(* Logix 5000 project; controller Safety vendor 1 type 14 code 86 rev 19.11; software revision 19.01 *)

TASK Periodic_0050ms (periodic, rate 50 ms, priority 11, watchdog 500 ms) : Comms
TASK SafetyTask (periodic, rate 50 ms, priority 10, watchdog 50 ms) : System, Estops, SafeOff

MODULES
   Local : vendor 1 type 14 code 86 (ICP 0, rev 19.11)
      Machine : vendor 1 type 14 code 96 (ICP 8, rev 19.13, $ae76c050$ RPI 20 ms)
      S16 : 1756-EN2T (Ethernet 192.168.1.200, ICP 16, rev 5.8)
      S2 : 1756-EN2T (ICP 2, Ethernet 192.168.1.10, rev 5.8, Input RPI 500 ms)
         SrDie_S1 : 1756-EN2T (Ethernet 192.168.1.18, rev 5.8)   // Shear Die Slot 01
            ShearDie : vendor 1 type 14 code 96 (ICP 0, rev 19.13, $8446c931$ RPI 20 ms)   // Shear Die Processor (Exit Section)
         CHPLC : 1734-AENTR (Ethernet 192.168.1.42, rev 3.10)
             : vendor 1 type 35 code 16 (PointIO 5, rev 1.1, Input RPI 50 ms, Output RPI 50 ms)
             : vendor 1 type 35 code 15 (PointIO 1, rev 1.1, Input RPI 50 ms)
             : vendor 1 type 35 code 15 (PointIO 3, rev 1.1, Input RPI 50 ms)
             : vendor 1 type 35 code 15 (PointIO 2, rev 1.1, Input RPI 50 ms)
             : vendor 1 type 35 code 16 (PointIO 6, rev 1.1, Input RPI 50 ms, Output RPI 50 ms)
             : vendor 1 type 35 code 16 (PointIO 4, rev 1.1, Output RPI 50 ms, Input RPI 50 ms)
         OS13 : 1734-AENTR (Ethernet 192.168.1.104, rev 3.10)
             : vendor 1 type 35 code 15 (PointIO 1, rev 1.1, Input RPI 50 ms)
         MCC2 : 1734-AENTR (Ethernet 192.168.1.41, rev 3.10)
             : vendor 1 type 35 code 16 (PointIO 1, rev 1.1, Output RPI 50 ms, Input RPI 10 ms)
             : vendor 1 type 35 code 16 (PointIO 2, rev 1.1, Input RPI 10 ms, Output RPI 50 ms)
         SDPLC : 1734-AENTR (Ethernet 192.168.1.79, rev 3.10)
             : vendor 1 type 35 code 15 (PointIO 1, rev 1.1, Input RPI 50 ms)
             : vendor 1 type 35 code 16 (PointIO 2, rev 1.1, Input RPI 50 ms, Output RPI 50 ms)
         MCC5 : 1734-AENTR (Ethernet 192.168.1.96, rev 3.10)
             : vendor 1 type 35 code 15 (PointIO 1, rev 1.1, Input RPI 10 ms)
             : vendor 1 type 35 code 16 (PointIO 5, rev 1.1, Input RPI 10 ms, Output RPI 50 ms)
             : vendor 1 type 35 code 16 (PointIO 3, rev 1.1, Input RPI 10 ms, Output RPI 50 ms)
             : vendor 1 type 35 code 16 (PointIO 4, rev 1.1, Input RPI 10 ms, Output RPI 50 ms)
         H1 : 1734-AENTR (Ethernet 192.168.1.120, rev 3.10)
             : vendor 1 type 35 code 15 (PointIO 6, rev 1.1, Input RPI 50 ms)
             : vendor 1 type 35 code 16 (PointIO 5, rev 1.1, Input RPI 50 ms, Output RPI 50 ms)
         G1 : 1734-AENTR (Ethernet 192.168.1.114, rev 3.10)
             : vendor 1 type 35 code 15 (PointIO 12, rev 1.1, Input RPI 50 ms)
             : vendor 1 type 35 code 16 (PointIO 11, rev 1.1, Input RPI 50 ms, Output RPI 50 ms)
         OS9 : 1734-AENTR (Ethernet 192.168.1.108, rev 3.10)
             : vendor 1 type 35 code 15 (PointIO 1, rev 1.1, Input RPI 50 ms)
         OS11 : 1734-AENTR (Ethernet 192.168.1.106, rev 3.10)
             : vendor 1 type 35 code 15 (PointIO 1, rev 1.1, Input RPI 50 ms)
         VS2 : 1734-AENTR (Ethernet 192.168.1.110, rev 3.10)
             : vendor 1 type 35 code 16 (PointIO 10, rev 1.1, Input RPI 50 ms, Output RPI 50 ms)
         OS16 : 1734-AENTR (Ethernet 192.168.1.97, rev 3.10)
             : vendor 1 type 35 code 15 (PointIO 1, rev 1.1, Input RPI 50 ms)
         OS8 : 1734-AENTR (Ethernet 192.168.1.116, rev 3.10)
             : vendor 1 type 35 code 15 (PointIO 1, rev 1.1, Input RPI 50 ms)
         E1 : 1734-AENTR (Ethernet 192.168.1.118, rev 3.10)
             : vendor 1 type 35 code 16 (PointIO 10, rev 1.1, Output RPI 50 ms, Input RPI 50 ms)
         DPD : 1734-AENTR (Ethernet 192.168.1.77, rev 3.10)
             : vendor 1 type 35 code 15 (PointIO 15, rev 1.1, Input RPI 50 ms)
             : vendor 1 type 35 code 16 (PointIO 14, rev 1.1, Input RPI 50 ms, Output RPI 50 ms)
         F1 : 1734-AENTR (Ethernet 192.168.1.112, rev 3.10)
             : vendor 1 type 35 code 15 (PointIO 20, rev 1.1, Input RPI 10 ms)
             : vendor 1 type 35 code 16 (PointIO 19, rev 1.1, Output RPI 50 ms, Input RPI 10 ms)
         OS14 : 1734-AENTR (Ethernet 192.168.1.102, rev 3.10)
             : vendor 1 type 35 code 15 (PointIO 1, rev 1.1, Input RPI 50 ms)
         MCC4 : 1734-AENTR (Ethernet 192.168.1.83, rev 3.10)
             : vendor 1 type 35 code 16 (PointIO 3, rev 1.1, Output RPI 50 ms, Input RPI 10 ms)
             : vendor 1 type 35 code 15 (PointIO 1, rev 1.1, Input RPI 10 ms)
             : vendor 1 type 35 code 16 (PointIO 4, rev 1.1, Output RPI 50 ms, Input RPI 10 ms)
         OS15 : 1734-AENTR (Ethernet 192.168.1.100, rev 3.10)
             : vendor 1 type 35 code 15 (PointIO 1, rev 1.1, Input RPI 50 ms)
      S3 : 1756-EN2T (Ethernet 192.168.1.11, ICP 3, rev 5.8, Input RPI 500 ms)
         OS3 : 1734-AENTR (Ethernet 192.168.1.40, rev 3.10)
             : vendor 1 type 35 code 15 (PointIO 1, rev 1.1, Input RPI 50 ms)
         OS1 : 1734-AENTR (Ethernet 192.168.1.70, rev 3.10)
             : vendor 1 type 35 code 15 (PointIO 1, rev 1.1, Input RPI 50 ms)
         D1 : 1734-AENTR (Ethernet 192.168.1.69, rev 3.10)
             : vendor 1 type 35 code 16 (PointIO 12, rev 1.1, Output RPI 50 ms, Input RPI 50 ms)
         OS4S : 1734-AENTR (Ethernet 192.168.1.57, rev 3.10)
             : vendor 1 type 35 code 16 (PointIO 5, rev 1.1, Input RPI 50 ms, Output RPI 50 ms)
             : vendor 1 type 35 code 15 (PointIO 1, rev 1.1, Input RPI 50 ms)
         OS5 : 1734-AENTR (Ethernet 192.168.1.62, rev 3.10)
             : vendor 1 type 35 code 15 (PointIO 1, rev 1.1, Input RPI 50 ms)
         A1 : 1734-AENTR (Ethernet 192.168.1.68, rev 3.10)
             : vendor 1 type 35 code 16 (PointIO 20, rev 1.1, Input RPI 50 ms, Output RPI 50 ms)
             : vendor 1 type 35 code 15 (PointIO 21, rev 1.1, Input RPI 50 ms)
         MCC3 : 1734-AENTR (Ethernet 192.168.1.38, rev 3.10)
             : vendor 1 type 35 code 16 (PointIO 4, rev 1.1, Input RPI 10 ms, Output RPI 50 ms)
             : vendor 1 type 35 code 16 (PointIO 3, rev 1.1, Input RPI 10 ms, Output RPI 50 ms)
             : vendor 1 type 35 code 15 (PointIO 1, rev 1.1, Input RPI 10 ms)
         MCC1 : 1734-AENTR (Ethernet 192.168.1.39, rev 3.10)
             : vendor 1 type 35 code 15 (PointIO 1, rev 1.1, Input RPI 10 ms)
             : vendor 1 type 35 code 16 (PointIO 6, rev 1.1, Input RPI 10 ms, Output RPI 50 ms)
         OS4N : 1734-AENTR (Ethernet 192.168.1.51, rev 3.10)
             : vendor 1 type 35 code 16 (PointIO 5, rev 1.1, Input RPI 50 ms, Output RPI 50 ms)
             : vendor 1 type 35 code 15 (PointIO 1, rev 1.1, Input RPI 50 ms)
         OS6 : 1734-AENTR (Ethernet 192.168.1.63, rev 3.10)
             : vendor 1 type 35 code 15 (PointIO 1, rev 1.1, Input RPI 50 ms)
         C1 : 1734-AENTR (Ethernet 192.168.1.43, rev 3.10)
             : vendor 1 type 35 code 16 (PointIO 12, rev 1.1, Output RPI 50 ms, Input RPI 10 ms)
         OS2 : 1734-AENTR (Ethernet 192.168.1.47, rev 3.10)
             : vendor 1 type 35 code 15 (PointIO 1, rev 1.1, Input RPI 50 ms)
      @b5ff5b04@:Partner : vendor 1 type 14 code 69 (ICP 1, rev 19.11)
END_MODULES

TYPE UDT_CardSts :
STRUCT
   EntrySts : DINT;   // Entry Status
   StandBy : BOOL;   // Stand By
   Faulted : BOOL;   // Faulted
   Validating : BOOL;   // Validating
   Connecting : BOOL;   // Connecting
   Running : BOOL;   // Running Connection OK
   ShuttingDown : BOOL;   // Shutting Down
   Inhibited : BOOL;   // Inhibited
   Waiting : BOOL;   // Waiting
END_STRUCT
END_TYPE

TYPE UDT_ShearStatus :
STRUCT
   Heartbeat : BOOL;   // Safety Status Heartbeat
   CoastStop : BOOL;   // Safety Status Coast Stop (0=Coast Stop) ( 1=OK)
   No_EStops : BOOL;   // Safety Status (0 = EStop) (1=OK)
   No_Faults : BOOL;   // Safety Status (1=No Faults)
   No_Motion : BOOL;   // Safety Status (1=No Motion)
   GuardsOK : BOOL;   // Safety Status Guards OK ( 1= OK)
   All_Drives_Off : BOOL;   // Safety Status All Drives Off (1=Off)
   ResetInput : BOOL;   // Safety Status Reset Input (1=Reset)
   FaultReset : BOOL;   // Safety Status (1=Fault Reset)
   CircuitReset : BOOL;   // Safety Status (1=Circuit Reset)
   CircuitResetTimer : TIMER;   // Safety Status Circuit Reset Timer
   StopTimer : TIMER;   // Safety Status Stop Timer Delay to Coast Drives
   BOOL : BOOL[32];   // Spare BOOLS
   DINT : DINT[5];   // Spare DINT
END_STRUCT
END_TYPE

TYPE UDT_SysStatus :
STRUCT
   Heartbeat : BOOL;   // Safety Status Heartbeat
   CoastStop_CTC : BOOL;   // Coil To Coil Safety Status Coast Stop (0=Coast Stop) ( 1=OK)
   CoastStop_CTL : BOOL;   // Cut To Length Safety Status Coast Stop (0=Coast Stop) ( 1=OK)
   CoastStop_Total : BOOL;   // Total Mode Safety Status Coast Stop (0=Coast Stop) ( 1=OK)
   No_CTC_EStops : BOOL;   // CTC Safety Status (0 = EStop) (1=OK)
   No_CTL_EStops : BOOL;   // CTL Safety Status (0 = EStop) (1=OK)
   No_Total_Estops : BOOL;   // Total Safety Status (0 = EStop) (1=OK)
   No_CTC_Faults : BOOL;   // Coil To Coil Safety Status (1=No Faults)
   No_CTL_Faults : BOOL;   // Cut To Length Safety Status (1=No Faults)
   No_Total_Faults : BOOL;   // Total Mode Safety Status (1=No Faults)
   No_Motion : BOOL;   // Safety Status (1=No Motion)
   GuardsOK : BOOL;   // Safety Status Guards OK ( 1= OK)
   All_Drives_Off : BOOL;   // Safety Status All Drives Off (1=Off)
   ResetInput_CTC : BOOL;   // Safety Status CTC Reset Input (1=Reset)
   ResetInput_CTL : BOOL;   // Safety Status CTL Reset Input (1=Reset)
   ResetInput_Total : BOOL;   // Safety Status Total Reset Input (1=Reset)
   FaultReset_CTC : BOOL;   // Safety Status CTC (1=Fault Reset)
   FaultReset_CTL : BOOL;   // Safety Status CTL (1=Fault Reset)
   FaultReset_Total : BOOL;   // Safety Status Total (1=Fault Reset)
   CircuitReset_CTC : BOOL;   // Safety Status CTC (1=Circuit Reset)
   CircuitReset_CTL : BOOL;   // Safety Status CTL (1=Circuit Reset)
   CircuitReset_Total : BOOL;   // Safety Status Total (1=Circuit Reset)
   CircuitResetTimer_CTC : TIMER;   // Safety Status Circuit Reset Timer
   CircuitResetTimer_CTL : TIMER;   // Safety Status CTL Circuit Reset Timer
   CircuitResetTimer_Total : TIMER;   // Safety Status Total Circuit Reset Timer
   CTCStopTimer : TIMER;   // Coil To Coil Safety Status Stop Timer Delay to Coast Drives
   CTLStopTimer : TIMER;   // Cut To Length Safety Status Stop Timer Delay to Coast Drives
   TotalStopTimer : TIMER;   // Total Mode Safety Status Stop Timer Delay to Coast Drives
   BOOL : BOOL[32];   // Spare BOOLS
   DINT : DINT[5];   // Spare DINT
END_STRUCT
END_TYPE

VAR_GLOBAL   (* controller tags *)
   A1_CoilCarSolPwrEn : BOOL;   // A1 UNW COIL CAR Solenoid Safe-Off Enable ( 1= Enable )
   A1_IO : UDT_CardSts[32] := ([0].EntrySts := 16897, [0].Running := 1);   // A1 Point I/O
        [4]   // 1734-IE2C/C
   A1_IOSts_Flt : BOOL;   // A1 Point IO Module Fault ( 1= Faulted)
   A1_S20_ModFlt : ALIAS FOR Flt_Modules[0].0;   // A1 Point I/O Slot20 Module Fault (1 = Fault)
   A1_S21_ModFlt : ALIAS FOR Flt_Modules[0].1;   // A1 Point I/O Slot21 Module Fault (1 = Fault)
   A1_SolPwrEn : BOOL := 1;   // A1 Solenoid Safe-Off Enable ( 1= Enable )
   A1_UnwLC_OK : BOOL := 1;   // Unwind Light Curtain A/B ( 1= Not Blocked) ( 0= Blocked)
   A1_UnwLC_RstCmd : BOOL;   // Unwind Light Curtain Reset Command ( 1= Reset Cmd)
   C1_IO : UDT_CardSts[32] := ([0].EntrySts := 16897, [0].Running := 1);   // C1 Point I/O
   C1_IOSts_Flt : BOOL;   // C1 Point IO Module Fault ( 1= Faulted)
   C1_S12_ModFlt : ALIAS FOR Flt_Modules[0].2;   // C1 Point I/O Slot12 Module Fault (1 = Fault)
   C1_SolPwrEn : BOOL := 1;   // C1 Solenoid Safe-Off Enable ( 1= Enable )
   CC : ALIAS FOR Diag_Tmp.0;   // Chris Como's Test Bit Always On Bit
   CC_Toggle : DINT := 4;   // TEST
   ChgMe : BOOL;
   ChgMe_x203PBL620 : BOOL;   // Need this from Machine OS1 Panel
   CHPLC_IO : UDT_CardSts[32] := ([0].EntrySts := 16897, [0].Running := 1);   // CHPLC Point I/O
   CHPLC_IOSts_Flt : BOOL;   // CHPLC Point IO Module Fault ( 1= Faulted)
   CHPLC_S1_ModFlt : ALIAS FOR Flt_Modules[0].3;   // CHPLC Point I/O Slot01 Module Fault (1 = Fault)
   CHPLC_S2_ModFlt : ALIAS FOR Flt_Modules[0].4;   // CHPLC Point I/O Slot02 Module Fault (1 = Fault)
   CHPLC_S3_ModFlt : ALIAS FOR Flt_Modules[0].5;   // CHPLC Point I/O Slot03 Module Fault (1 = Fault)
   CHPLC_S4_ModFlt : ALIAS FOR Flt_Modules[0].6;   // CHPLC Point I/O Slot04 Module Fault (1 = Fault)
   CHPLC_S5_ModFlt : ALIAS FOR Flt_Modules[0].7;   // CHPLC Point I/O Slot05 Module Fault (1 = Fault)
   CHPLC_S6_ModFlt : ALIAS FOR Flt_Modules[0].8;   // CHPLC Point I/O Slot06 Module Fault (1 = Fault)
   Citect_HB_Flt : BOOL;   // Citect Heartbeat Fault ( 1= Fault)
   Citect_HB_TOF : TIMER := (PRE := 2000, EN := 1, DN := 1);   // Citect Heartbeat Timer Off
   Citect_HB_TON : TIMER := (PRE := 2000, ACC := 850, EN := 1, TT := 1);   // Citect Heartbeat Timer On
   CommCards_OK : DINT := 30;   // Comm Cards OK
        .1   // Op Stations (Entry Section) Comm Cards OK ( 1= OK)
        .0   // MCC Comm Cards OK ( 1= OK)
        .2   // Op Stations (Exit Section) Comm Cards OK ( 1= OK)
        .3   // General I/O Comm Cards OK ( 1= OK)
        .4   // General I/O Comm Cards OK ( 1= OK)
        .31   // ALL Comm Cards OK ( 1= OK)
   D1_IO : UDT_CardSts[32] := ([0].EntrySts := 16897, [0].Running := 1);   // D1 Point I/O
        [4]   // 1734-IE2C/C
   D1_IOSts_Flt : BOOL;   // D1 Point IO Module Fault ( 1= Faulted)
   D1_S12_ModFlt : ALIAS FOR Flt_Modules[0].9;   // D1 Point I/O Slot12 Module Fault (1 = Fault)
   D1_SolPwrEn : BOOL := 1;   // D1 Solenoid Safe-Off Enable ( 1= Enable )
   DAM : ALIAS FOR Diag_Tmp.4;   // Doug M Always Off Test Bit
   Daniel_Ponstein_AFI : BOOL;
   Darin_M_Safety_Test_Bit : BOOL := 1;
   Darin_M_Test_Bit : DINT;
   DavidTest : BOOL;
   Diag_Tmp : DINT := 4079;   // Temp Bit Test Bit
        .17   // Temporary Test Bit: Logic 17
        .18   // Temporary Test Bit: Logic 18
        .0   // Temporary Test Bit 0: Logic 1
        .1   // Temporary Test Bit 1: Logic 1
        .10   // Temporary Test Bit: Logic 10
        .11   // Temporary Test Bit: Logic 11
        .12   // Temporary Test Bit: Logic 12
        .13   // Temporary Test Bit: Logic 13
        .14   // Temporary Test Bit: Logic 14
        .15   // Temporary Test Bit: Logic 15
        .16   // Temporary Test Bit: Logic 16
        .19   // Temporary Test Bit: Logic 19
        .2   // Temporary Test Bit 2: Logic 1
        .20   // Temporary Test Bit: Logic 20
        .21   // Temporary Test Bit: Logic 21
        .22   // Temporary Test Bit: Logic 22
        .23   // Temporary Test Bit: Logic 23
        .24   // Temporary Test Bit: Logic 24
        .25   // Temporary Test Bit: Logic 25
        .26   // Temporary Test Bit: Logic 26
        .27   // Temporary Test Bit: Logic 27
        .28   // Temporary Test Bit: Logic 28
        .29   // Temporary Test Bit: Logic 29
        .3   // Temporary Test Bit 3: Logic 1
        .30   // Temporary Test Bit: Logic 30
        .31   // Temporary Test Bit: Logic 31
        .4   // Temporary Test Bit 4: Logic 1
        .5   // Temporary Test Bit 5: Logic 1
        .6   // Temporary Test Bit 6: Logic 1
        .7   // Temporary Test Bit 6: Logic 1
        .8   // Temporary Test Bit: Logic 8
        .9   // Temporary Test Bit: Logic 9
   DPD_EstopRstCmd : BOOL;   // DPD Estop Reset Cmd
   DPD_FltRstCmd : BOOL;   // DPD Fault Reset Cmd
   DPD_IO : UDT_CardSts[32] := ([0].EntrySts := 16897, [0].Running := 1);   // DPD Point I/O
        [4]   // 1734-IE2C/C
   DPD_IOSts_Flt : BOOL;   // DPD Point IO Module Fault ( 1= Faulted)
   DPD_No_EStops : BOOL := 1;   // DPD No Estops ( 1= OK)
   DPD_S14_ModFlt : ALIAS FOR Flt_Modules[0].10;   // DPD Point I/O Slot14 Module Fault (1 = Fault)
   DPD_S15_ModFlt : ALIAS FOR Flt_Modules[0].11;   // DPD Point I/O Slot15 Module Fault (1 = Fault)
   DPD_SolPwrEn : BOOL := 1;   // DPD Solenoid Safe-Off Enable ( 1= Enable )
   Drives_Off : DINT;   // Line Drives Off
        .1   // Line AC Drives Off ( 1= Drvs Off)
        .0   // Line All DC Drives Off ( 1= Drvs Off)
        .4   // Shear Die Accelerator Drives Off ( 1= Drvs Off)
        .2   // Line AC Drives Off ( 1= Drvs Off)
        .3   // Line AC Drives Off ( 1= Drvs Off)
   E1_IO : UDT_CardSts[32] := ([0].EntrySts := 16897, [0].Running := 1);   // E1 Point I/O
        [4]   // 1734-IE2C/C
   E1_IOSts_Flt : BOOL;   // E1 Point IO Module Fault ( 1= Faulted)
   E1_S10_ModFlt : ALIAS FOR Flt_Modules[0].12;   // E1 Point I/O Slot10 Module Fault (1 = Fault)
   E1_SolPwrEn : BOOL := 1;   // E1 Solenoid Safe-Off Enable ( 1= Enable )
   EnBridle_DrvsOff : BOOL;   // Entry Bridle Drives OFF ( 1= OFF)
   EnBridle_SafeOffEn : BOOL := 1;   // Entry Bridle Safe-Off Enable ( 1= Enable )
   EnBridle_SafeOffFltRst : BOOL;   // Entry Bridle Safe-Off Fault Reset ( 1= Reset Cmd )
   ES_IndJog_PB : BOOL;   // Exit Section Individual Jog Select ( 1= Req Individual)
   ES_Line_JogPB : BOOL;   // Exit Section Line Jog PB ( 1= Ind Jog )
   ES_Line_RunPB : BOOL;   // Exit Section Line Run PB ( 1= Run)
   ES_Line_StopPB : BOOL := 1;   // Exit Section Line Stop PB ( 1= OK) (0=Stop)
   ES_Line_ThreadPB : BOOL;   // Exit Section Line Thread PB ( 1= Thread)
   ES_TndJog_PB : BOOL;   // Exit Section Tandem Jog PB (1= Tandem Jog Sel)
   ESTOP_x201PB040 : DCI_STOP := (ChannelA := 1, ChannelB := 1, InputStatus := 1, ColdStartType := 1, DiscrepancyTime := 250, O1 := 1);   // OS1 Line EStop Pushbutton
   ESTOP_x201PB040_Flt : ALIAS FOR Flt_Estops.0;   // OS1 Line EStop Pushbutton Fault ( 1= Fault)
   ESTOP_x211PB040 : DCI_STOP := (ChannelA := 1, ChannelB := 1, InputStatus := 1, ColdStartType := 1, DiscrepancyTime := 250, O1 := 1);   // OS2 Line EStop Pushbutton
   ESTOP_x211PB040_Flt : ALIAS FOR Flt_Estops.1;   // OS2 Line EStop Pushbutton Fault ( 1= Fault)
   ESTOP_x221PB040 : DCI_STOP := (ChannelA := 1, ChannelB := 1, InputStatus := 1, ColdStartType := 1, DiscrepancyTime := 250, O1 := 1);   // OS3 Line EStop Pushbutton
   ESTOP_x221PB040_Flt : ALIAS FOR Flt_Estops.2;   // OS3 Line EStop Pushbutton Fault ( 1= Fault)
   ESTOP_x231PB040 : DCI_STOP := (ChannelA := 1, ChannelB := 1, InputStatus := 1, ColdStartType := 1, DiscrepancyTime := 250, O1 := 1);   // OS4N Line EStop Pushbutton
   ESTOP_x231PB040_Flt : ALIAS FOR Flt_Estops.3;   // OS4N Line EStop Pushbutton Fault ( 1= Fault)
   ESTOP_x241PB040 : DCI_STOP := (ChannelA := 1, ChannelB := 1, InputStatus := 1, ColdStartType := 1, DiscrepancyTime := 250, O1 := 1);   // OS4S Line EStop Pushbutton
   ESTOP_x241PB040_Flt : ALIAS FOR Flt_Estops.4;   // OS4S Line EStop Pushbutton Fault ( 1= Fault)
   ESTOP_x251PB040 : DCI_STOP := (ChannelA := 1, ChannelB := 1, InputStatus := 1, ColdStartType := 1, DiscrepancyTime := 250, O1 := 1);   // OS5 Line EStop Pushbutton
   ESTOP_x251PB040_Flt : ALIAS FOR Flt_Estops.5;   // OS5 Line EStop Pushbutton Fault ( 1= Fault)
   ESTOP_x261PB040 : DCI_STOP := (ChannelA := 1, ChannelB := 1, InputStatus := 1, ColdStartType := 1, DiscrepancyTime := 250, O1 := 1);   // OS6 Line EStop Pushbutton
   ESTOP_x261PB040_Flt : ALIAS FOR Flt_Estops.6;   // OS6 Line EStop Pushbutton Fault ( 1= Fault)
   ESTOP_x271PB040 : DCI_STOP := (ChannelA := 1, ChannelB := 1, InputStatus := 1, ColdStartType := 1, DiscrepancyTime := 250, O1 := 1);   // OS8 Line EStop Pushbutton
   ESTOP_x271PB040_Flt : ALIAS FOR Flt_Estops.7;   // OS8 Line EStop Pushbutton Fault ( 1= Fault)
   ESTOP_x281PB040 : DCI_STOP := (ChannelA := 1, ChannelB := 1, InputStatus := 1, ColdStartType := 1, DiscrepancyTime := 250, O1 := 1);   // OS9 Line EStop Pushbutton
   ESTOP_x281PB040_Flt : ALIAS FOR Flt_Estops.8;   // OS9 Line EStop Pushbutton Fault ( 1= Fault)
   ESTOP_x291PB040 : DCI_STOP := (ChannelA := 1, ChannelB := 1, InputStatus := 1, ColdStartType := 1, DiscrepancyTime := 250, O1 := 1);   // OS11 Line EStop Pushbutton
   ESTOP_x291PB040_Flt : ALIAS FOR Flt_Estops.9;   // OS11 Line EStop Pushbutton Fault ( 1= Fault)
   ESTOP_x301PB040 : DCI_STOP := (ChannelA := 1, ChannelB := 1, InputStatus := 1, ColdStartType := 1, DiscrepancyTime := 250, O1 := 1);   // OS13 Line EStop Pushbutton
   ESTOP_x301PB040_Flt : ALIAS FOR Flt_Estops.10;   // OS13 Line EStop Pushbutton Fault ( 1= Fault)
   ESTOP_x311PB040 : DCI_STOP := (ChannelA := 1, ChannelB := 1, InputStatus := 1, ColdStartType := 1, DiscrepancyTime := 250, O1 := 1);   // OS14 Line EStop Pushbutton
   ESTOP_x311PB040_Flt : ALIAS FOR Flt_Estops.11;   // OS14 Line EStop Pushbutton Fault ( 1= Fault)
   ESTOP_x311PB130 : DCI_STOP := (ChannelA := 1, ChannelB := 1, InputStatus := 1, ColdStartType := 1, DiscrepancyTime := 250, O1 := 1);   // OS14 Shear Estop Pushbutton
   ESTOP_x311PB130_Flt : ALIAS FOR Flt_Estops.17;   // OS14 Shear EStop Pushbutton Fault ( 1= Fault)
   ESTOP_x321PB040 : DCI_STOP := (ChannelA := 1, ChannelB := 1, InputStatus := 1, ColdStartType := 1, DiscrepancyTime := 250, O1 := 1);   // OS15 Line EStop Pushbutton
   ESTOP_x321PB040_Flt : ALIAS FOR Flt_Estops.12;   // OS15 Line EStop Pushbutton Fault ( 1= Fault)
   ESTOP_x331PB040 : DCI_STOP := (ChannelA := 1, ChannelB := 1, InputStatus := 1, ColdStartType := 1, DiscrepancyTime := 250, O1 := 1);   // OS16 Line EStop Pushbutton
   ESTOP_x331PB040_Flt : ALIAS FOR Flt_Estops.13;   // OS16 Line EStop Pushbutton Fault ( 1= Fault)
   ESTOP_x480PB470 : DCI_STOP := (ChannelA := 1, ChannelB := 1, InputStatus := 1, ColdStartType := 1, DiscrepancyTime := 250, O1 := 1);   // DPD Line EStop Pushbutton
   ESTOP_x480PB470_Flt : ALIAS FOR Flt_Estops.14;   // DPD Line EStop Pushbutton Fault ( 1= Fault)
   ESTOP_x480PB550 : DCI_STOP := (ChannelA := 1, ChannelB := 1, InputStatus := 1, ColdStartType := 1, DiscrepancyTime := 250, O1 := 1);   // DPD (In Pit) Line EStop Pushbutton
   ESTOP_x480PB550_Flt : ALIAS FOR Flt_Estops.15;   // DPD Line EStop Pushbutton Fault ( 1= Fault)
   ESTOP_x519LS470 : DCI_STOP := (ChannelA := 1, ChannelB := 1, InputStatus := 1, ColdStartType := 1, DiscrepancyTime := 250, O1 := 1);   // G1 Tripwire Line EStop
   ESTOP_x519LS470_Flt : ALIAS FOR Flt_Estops.18;   // G1 Line EStop Tripwire Limit Switch Fault ( 1= Fault)
   ESTOP_x533PB470 : DCI_STOP := (ChannelA := 1, ChannelB := 1, InputStatus := 1, ColdStartType := 1, DiscrepancyTime := 250, O1 := 1);   // H1 Line EStop Pushbutton
   ESTOP_x533PB470_Flt : ALIAS FOR Flt_Estops.16;   // H1 Line EStop Pushbutton Fault ( 1= Fault)
   ExBridle_DrvsOff : BOOL;   // Exit Bridle Drives OFF ( 1= OFF)
   ExBridle_SafeOffEn : BOOL := 1;   // Exit Bridle Safe-Off Enable ( 1= Enable )
   ExBridle_SafeOffFltRst : BOOL;   // Exit Bridle Safe-Off Fault Reset ( 1= Reset Cmd )
   ExConHydPump_AutoStart : BOOL;   // (From Mach) Exit Conveyor Hydraulic Pump Auto Start Command
   F1_CoilCarSolPwrEn : BOOL := 1;   // F1 UNW COIL CAR Solenoid Safe-Off Enable ( 1= Enable )
   F1_IO : UDT_CardSts[32] := ([0].EntrySts := 16897, [0].Running := 1);   // F1 Point I/O
        [4]   // 1734-IE2C/C
   F1_IOSts_Flt : BOOL;   // F1 Point IO Module Fault ( 1= Faulted)
   F1_S19_ModFlt : ALIAS FOR Flt_Modules[0].13;   // F1 Point I/O Slot19 Module Fault (1 = Fault)
   F1_S20_ModFlt : ALIAS FOR Flt_Modules[0].14;   // F1 Point I/O Slot20 Module Fault (1 = Fault)
   F1_SolPwrEn : BOOL := 1;   // F1 Solenoid Safe-Off Enable ( 1= Enable )
   Flattener_FVR_En : BOOL := 1;   // Flattener FVR Enable ( 1= Enable )
   Flattener_FVR_FltRst : BOOL;   // Flattener Fault Reset ( 1= Reset Cmd )
   Flattener_FVR_FwdCmd : BOOL;   // Flattener Forward Command ( 1= Run Fwd )
   Flattener_FVR_RevCmd : BOOL;   // Flattener Reverse Command ( 1= Run Rev)
   Flt_Estops : DINT;   // Estop Fault Word
   Flt_Modules : DINT[5];   // Point IO Module Fault Word
   Flt_SafeOff : DINT[3];   // Safe Off Fault Word
   Flt_Starter : DINT;   // Starter Fault Word
   FltsToCitect : DINT[64];   // Faults to Citect
        [2]   // (Faults to Citect) Estop PB Faults
        [3]   // (Faults to Citect) Safe-Off Relay Faults
        [4]   // (Faults to Citect) FVR/FVNR Starter Faults
        [7]   // (Faults to Citect) MCC I/O Safety Module Faults
        [1]   // (Faults to Citect) Remote I/O Comm Faults
        [5]   // (Faults to Citect) General I/O Safety Module Faults
        [6]   // (Faults to Citect) Operator Station I/O Safety Module Faults
        [0].0   // Comm Loss Machine PLC
        [0].1   // Comm Loss Shear Die PLC
        [0].3   // Comm Loss Safety Slot 2
        [0].4   // Comm Loss Safety Slot 3
        [0].5   // Comm Loss Safety Slot 16
   FromCitect : DINT[64] := ([0] := 1, [10] := 22000, [11] := 22000, [12] := 12000, [13] := 12000, [14] := 12000);   // (From Citect)
        [1].10   // (From Citect)
        [1].12   // (From Citect)
        [1].13   // (From Citect)
        [1].14   // (From Citect)
        [1].15   // (From Citect)
        [1].16   // (From Citect)
        [1].11   // (From Citect)
        [0].19   // (From Citect)
        [0].0   // (From Citect) Heartbeat Reflected Back
        [0].1   // (From Citect) Exit Conveyor Hyd Pump Start
        [0].10   // (From Citect) Neg Tolerance Load PB
        [0].11   // (From Citect) Warning Count Load PB
        [0].12   // (From Citect) Scrap Length Load PB
        [0].13   // (From Citect) Scrap Reset PB
        [0].14   // (From Citect) Skid Count Load PB
        [0].15   // (From Citect) Shear Crank Start PB
        [0].16   // (From Citect) Shear Crank Stop PB
        [0].17   // (From Citect) Product Conveyors Start Command PB ( 1= Start)
        [0].18   // (From Citect) Product Conveyors Stop Command PB ( 1= Stop)
        [0].2   // (From Citect) Exit Conveyor Hyd Pump Stop
        [0].20   // (From Citect) Shear Pinch Roll Short Loop Select ( 1= Short Loop )
        [0].21   // (From Citect) Shear Pinch Roll Long Loop Select ( 1= Short Loop )
        [0].22   // (From Citect) Stacker Counter Reset PB
        [0].23   // (From Citect) Stacker Counter Increment PB
        [0].24   // (From Citect) Stacker Counter Decrement PB
        [0].25   // (From Citect) Good Piece Counter Reset PB
        [0].26   // (From Citect) Good Piece Counter Increment PB
        [0].27   // (From Citect) Good Piece Counter Decrement PB
        [0].28   // (From Citect) Lot Good Piece Counter Reset PB
        [0].29   // (From Citect) Lot Good Piece Counter Increment PB
        [0].3   // (From Citect) Sheeter Hyd Pump Start
        [0].30   // (From Citect) Lot Good Piece Counter Decrement PB
        [0].31   // (From Citect) Scrap Piece Counter Reset PB
        [0].4   // (From Citect) Sheeter Hyd Pump Stop
        [0].5   // (From Citect) Cut Length Load PB
        [0].6   // (From Citect) Cut Length Increase PB
        [0].7   // (From Citect) Cut Length Decrease PB
        [0].8   // (From Citect) Sheet Count Load PB
        [0].9   // (From Citect) Pos Tolerance Load PB
        [1].0   // (From Citect) Scrap Piece Counter Increment PB
        [1].1   // (From Citect) Scrap Piece Counter Decrement PB
        [1].17   // (From Citect)
        [1].18   // (From Citect)
        [1].19   // (From Citect)
        [1].2   // (From Citect) Home Position Set Command ( 1= Set Home Pos)
        [1].20   // (From Citect)
        [1].21   // (From Citect)
        [1].22   // (From Citect)
        [1].23   // (From Citect)
        [1].24   // (From Citect)
        [1].25   // (From Citect)
        [1].26   // (From Citect)
        [1].27   // (From Citect)
        [1].28   // (From Citect)
        [1].29   // (From Citect)
        [1].3   // (From Citect) Shear Lube Pump Start Command
        [1].30   // (From Citect)
        [1].31   // (From Citect)
        [1].4   // (From Citect) Shear Lube Pump Stop Command
        [1].5   // (From Citect) Sheeter Lube Pump Start Command
        [1].6   // (From Citect) Sheeter Lube Pump Stop Command
        [1].7   // (From Citect) Shear Metering Back Up Roll Light Gage Select
        [1].8   // (From Citect) Shear Metering Back Up Roll Heavy Gage Select
        [1].9   // (From Citect)
        [2].0   // (From Citect)
        [2].1   // (From Citect)
        [2].10   // (From Citect)
        [2].11   // (From Citect)
        [2].12   // (From Citect)
        [2].13   // (From Citect)
        [2].14   // (From Citect)
        [2].15   // (From Citect)
        [2].16   // (From Citect)
        [2].17   // (From Citect)
        [2].18   // (From Citect)
        [2].19   // (From Citect)
        [2].2   // (From Citect)
        [2].20   // (From Citect)
        [2].21   // (From Citect)
        [2].22   // (From Citect)
        [2].23   // (From Citect)
        [2].24   // (From Citect)
        [2].25   // (From Citect)
        [2].26   // (From Citect)
        [2].27   // (From Citect)
        [2].28   // (From Citect)
        [2].29   // (From Citect)
        [2].3   // (From Citect)
        [2].30   // (From Citect)
        [2].31   // (From Citect)
        [2].4   // (From Citect)
        [2].5   // (From Citect)
        [2].6   // (From Citect)
        [2].7   // (From Citect)
        [2].8   // (From Citect)
        [2].9   // (From Citect)
        [3]   // (From Citect) Set Scrap Length Inch
        [4]   // (From Citect) Warning Count
        [5]   // (From Citect) Next Cut Length Inch
        [6]   // (From Citect) Neg Tolerance Setpoint
        [7]   // (From Citect) Cut Length Inch
        [8]   // (From Citect) Skid Count Setpoint Pieces/Skid
        [9]   // (From Citect) Sheet Count Setpoint Pieces Before Warning
   FromMach : DINT[35];   // (FromMach)
   FromMachine : DINT[35] := ([0] := 164, [1] := 3, [3] := 16, [5] := 64, [10] := 50000, [11] := 100000, [12] := 1000000, [13] := 5000000, [15] := 3278258, [16] := 32, [19] := 44810, [21] := 44810);   // (FromMach)
        [0].1   // (FromMach) UWCC_Rst_PB Unwind Coil Car Safety Reset PB
        [0].24   // (FromMach)
        [0].25   // (FromMach)
        [0].7   // (FromMach)
        [0].4   // (FromMach)
        [0].3   // (FromMach)
        [0].0   // (FromMach) HB Heart Beat 0.25 Secs
        [0].19   // (FromMach)
        [0].20   // (FromMach)
        [0].21   // (FromMach)
        [0].23   // (FromMach)
        [0].18   // (FromMach)
        [0].8   // (FromMach)
        [0].9   // (FromMach)
        [0].16   // (FromMach)
        [0].17   // (FromMach)
        [0].22   // (FromMach)
        [0].5   // (FromMach)
        [0].10   // (FromMach) Hydraulic Pumps Auto Start Active
        [0].11   // (FromMach) Exit Conveyor Hydraulic Pump Auto Start Command
        [0].12   // (FromMach) Sheeter Hydraulic Pump Auto Start Command
        [0].13   // (FromMach) Lube Pumps Auto Start Active
        [0].14   // (FromMach) Sheeter PR Lube Pump Auto Start Command
        [0].15   // (FromMach) Shear PR Lube Pump Auto Start Command
        [0].26   // (FromMach)
        [0].27   // (FromMach)
        [0].28   // (FromMach)
        [0].29   // (FromMach)
        [0].30   // (FromMach)
        [0].31   // (FromMach)
        [1].0   // (FromMach)
        [1].1   // (FromMach)
        [1].2   // (FromMach)
        [1].3   // (FromMach)
        [1].4   // (FromMach)
        [1].5   // (FromMach)
        [1].6   // (FromMach)
        [1].7   // (FromMach)
        [1].8   // (FromMach)
        [1].9   // (FromMach)
        [1].10   // (FromMach)
        [1].11   // (FromMach)
        [1].12   // (FromMach)
        [1].13   // (FromMach)
        [1].14   // (FromMach)
        [1].15   // (FromMach)
        [1].16   // (FromMach)
        [1].17   // (FromMach)
        [1].18   // (FromMach)
        [1].19   // (FromMach)
        [1].20   // (FromMach)
        [1].21   // (FromMach)
        [1].22   // (FromMach)
        [1].23   // (FromMach)
        [1].24   // (FromMach)
        [1].25   // (FromMach)
        [1].26   // (FromMach)
        [1].27   // (FromMach)
        [1].28   // (FromMach)
        [1].29   // (FromMach)
        [1].30   // (FromMach)
        [1].31   // (FromMach)
        [2]   // (FromMach)
        [3]   // (FromMach)
        [4]   // (FromMach)
        [5].0   // (FromMach) Unwind Holddown Roll Jog Forward Command
        [5].1   // (FromMach) Unwind Holddown Roll Jog Reverse Command
        [5].2   // (FromMach) Flattener Jog Forward Command
        [5].3   // (FromMach) Flattener Jog Reverse Command
        [5].4   // (FromMach) Trimmer Pinch Roll Jog Forward Command
        [5].5   // (FromMach) Trimmer Pinch Roll Jog Reverse Command
        [5].6   // (FromMach) Trimmer Scrap Conveyor Jog Command
        [5].7   // (FromMach) Rewind Pinch Roll Jog Forward Command
        [5].8   // (FromMach) Rewind Pinch Roll Jog Reverse Command
        [5].9   // (FromMach)
        [5].10   // (FromMach)
        [5].11   // (FromMach)
        [5].12   // (FromMach)
        [5].13   // (FromMach)
        [5].14   // (FromMach)
        [5].15   // (FromMach)
        [5].16   // (FromMach)
        [5].17   // (FromMach)
        [5].18   // (FromMach)
        [5].19   // (FromMach)
        [5].20   // (FromMach)
        [5].21   // (FromMach)
        [5].22   // (FromMach)
        [5].23   // (FromMach)
        [5].24   // (FromMach)
        [5].25   // (FromMach)
        [5].26   // (FromMach)
        [5].27   // (FromMach)
        [5].28   // (FromMach)
        [5].29   // (FromMach)
        [5].30   // (FromMach)
        [5].31   // (FromMach)
        [0].6   // (FromMach) Line Emergency Stop Reset PBL
        [0].2   // (FromMach) Line TOTAL Mode ( 1= Total Mode) (0 = Coil to Coil)
   FromSafety : DINT[35] := ([0] := 16142, [1] := 14, [2] := 536870911, [4] := 64, [5] := 1); {produced}   // (From Safety)
        [2].30   // (From Safety)
        [0].0   // (From Safety) Heartbeat Pulse
        [5].0   // (From Safety) Shear Die Crank Running Fdbk ( 1= Running)
        [2].29   // (From Safety)
        [5].3   // (From Safety) Stacker Chain Fwd Fdbk
        [5].4   // (From Safety) Stacker Chain Rev Fdbk
        [5].1   // (From Safety) Scrap Horizontal Conveyor Fwd Fdbk
        [5].2   // (From Safety) Scrap Horizontal Conveyor Rev Fdbk
        [5].5   // (From Safety) Stacker Side Guide Lift Fwd Fdbk/Up
        [5].6   // (From Safety) Stacker Side Guide Lift Rev Fdbk/Down
        [4].3   // (From Safety) Flattener Drive Motor Rev Fdbk
        [1].1   // (From Safety) Shear Safety Status Coast Stop ( 0 = Coast Stop) ( 1= OK)
        [0].1   // (From Safety) Line Safety Status Coast Stop ( 0 = Coast Stop) ( 1= OK)
        [1].3   // (From Safety) Shear Safety Status No Faults ( 0 = Faults) ( 1= OK)
        [0].6   // (From Safety) Line Safety Status Guards OK ( 1= OK)
        [0]   // (From Safety)
        [0].8   // (From Safety)
        [0].4   // (From Safety)
        [0].9   // (From Safety)
        [0].7   // (From Safety)
        [2]   // (From Safety)
        [1].4   // (From Safety)
        [1].7   // (From Safety)
        [0].5   // (From Safety) Line Safety Status All Drives Off ( 1= All Off)
        [4].1   // (From Safety) Unwind Holddown Roll Drive Motor Rev Fdbk
        [0].2   // (From Safety) Line Safety Status EStop ( 0 = EStop) ( 1= OK)
        [0].3   // (From Safety) Line Safety Status No Faults ( 0 = Faults) ( 1= OK)
        [1].2   // (From Safety) Shear Safety Status EStop ( 0 = EStop) ( 1= OK)
        [1].5   // (From Safety) Shear Safety Status All Drives Off ( 1= All Off)
        [1].6   // (From Safety)
        [2].31   // (From Safety)
        [4].0   // (From Safety) Unwind Holddown Roll Drive Motor Fwd Fdbk
        [4].2   // (From Safety) Flattener Drive Motor Fwd Fdbk
        [4].4   // (From Safety) Trimmer Pinch Roll Fwd Fdbk
        [4].5   // (From Safety) Trimmer Pinch Roll Rev Fdbk
        [4].6   // (From Safety) Trimmer Scrap Conveyor RunFdbk
        [4].7   // (From Safety) Rewind Pinch Roll Fwd Fdbk
        [4].8   // (From Safety) Rewind Pinch Roll Rev Fdbk
        [2].0   // (From Safety) Unwind Op Side Drive Enable Relay
        [2].1   // (From Safety) Unwind Drive Side Drive Enable Relay
        [2].6   // (From Safety) Rewind Drive Enable Relay
        [2].9   // (From Safety) Paper Winder Safety Enable
        [2].12   // (From Safety) Scrap Choppers Safety Enable
        [2].22   // (From Safety) Shear Conveyor Safety Enable
        [2].27   // (From Safety) Stacker Blower Safety Enable
        [2].2   // (From Safety) #1 Entry Bridle Roll 2 Drive Enable Relay
        [2].3   // (From Safety) #2 Entry Bridle Roll 3 Drive Enable Relay
        [2].4   // (From Safety) #1 Exit Bridle Roll 6 Drive Enable Relay
        [2].5   // (From Safety) #2 Exit Bridle Roll 7 Drive Enable Relay
        [2].7   // (From Safety) Shear Die Drive Enable Relay
        [2].8   // (From Safety) Unwind Pinch Roll Safety Enable
        [2].10   // (From Safety) Trimmer Knives Width Adjust Safety Enable
        [2].11   // (From Safety) Trimmer Knives Safety Enable
        [2].13   // (From Safety) Scrap Choppers Width Adjust Safety Enable
        [2].14   // (From Safety) Washtank Pinch Roll 1 Safety Enable
        [2].15   // (From Safety) Washtank Pinch Roll 2 Safety Enable
        [2].16   // (From Safety) Washtank Pinch Roll 3 Safety Enable
        [2].17   // (From Safety) Washtank Pinch Roll 4 Safety Enable
        [2].18   // (From Safety) Side Guide Width Adjust Safety Enable
        [2].19   // (From Safety) Sheeter Pinch Roll Safety Enable
        [2].20   // (From Safety) Shear Pinch Roll Safety Enable
        [2].21   // (From Safety) Shear Metering Backup Roll Safety Enable
        [2].23   // (From Safety) Product Conveyor 1 Safety Enable
        [2].24   // (From Safety) Product Conveyor 2 Safety Enable
        [2].25   // (From Safety) Product Conveyor 3 Safety Enable
        [2].26   // (From Safety) Scrap Incline Conveyor Safety Enable
        [2].28   // (From Safety) Stacker Back Stop Safety Enable
   FromShearDie : DINT[35] := ([0] := 159, [1] := 8, [2] := 1056767, [5] := 1, [10] := 144000);   // (From Shear Die)
        [0].0   // (From Shear Die) Heartbeat Pulse
        [0].5   // (From Shear Die) Shear Emergency Stop Reset PBL
        [0].7   // (From Shear Die) Exit Section Line Stop PB ( 1= OK) (0=Stop)
        [0].10   // (From Shear Die) Exit Section Line Jog PB ( 1= Ind Jog)
        [5].3   // (From Shear Die) Stacker Chain Fwd Cmd
        [5].4   // (From Shear Die) Stacker Chain Rev Cmd
        [0].6   // (From Shear Die) Line Emergency Stop Reset PBL
        [0].4   // (From Shear DIe) Sheeter Pinch Roll Lube Run Fdbk
        [0].15   // (From Shear Die) Sheeter Pinch Roll Jog Forward SS
        [0].9   // (From Shear Die) Exit Section Line Thread PB ( 1= Thread)
        [0].8   // (From Shear Die) Exit Section Line Run PB ( 1= Run)
        [0].11   // (From Shear Die) Exit Section Tandem Jog PB (1= Tandem Jog Sel)
        [0].16   // (From Shear Die) Sheeter Pinch Roll Jog Reverse SS
        [0].1   // (From Shear DIe) Exit Conveyor Hyd Pump Run Fdbk
        [0].13   // (From Shear Die) Sheeter Pinch Roll Jog Forward SS
        [0].2   // (From Shear DIe) Sheeter Hyd Pump Run Fdbk
        [0].12   // (From Shear Die) Exit Section Individual Jog PB (1= Indiv Jog Sel)
        [0].18   // (From Shear Die) Shear Pinch Roll Jog Reverse SS
        [0].17   // (From Shear Die) Shear Pinch Roll Jog Forward SS
        [0].3   // (From Shear DIe) Shear Pinch Roll Lube Run Fdbk
        [0].14   // (From Shear Die) Sheeter Pinch Roll Jog Reverse SS
        [0].19   // (From Shear Die) Shear Conveyor Jog Forward SS
        [0].20   // (From Shear Die) Shear Conveyor Jog Reverse SS
        [0].21   // (From Shear Die) Product Conveyor Jog Forward PB
        [0].22   // (From Shear Die) Product Conveyor Jog Reverse PB
        [0].23   // (From Shear Die) Scrap Conveyor Jog Forward SS
        [0].24   // (From Shear Die) Scrap Conveyor Jog Reverse SS
        [1].0   // (From Shear Die) Scrap Mode Selected ( 1= Requested)
        [5].0   // (From Shear Die) Shear Die Crank Run Command ( 1= Run)
        [5].1   // (From Shear Die) Scrap Horizontal Conveyor Fwd Cmd ( 1= Run Fwd)
        [5].2   // (From Shear Die) Scrap Horizontal Conveyor Rev Cmd ( 1= Run Rev)
        [5].5   // (From Shear Die) Stacker Side Guide Lift Fwd Cmd/Up
        [5].6   // (From Shear Die) Stacker Side Guide Lift Rev Cmd/Dwn
   FUTURE : ALIAS FOR Diag_Tmp.1;   // FUTURE
   FVNR_y761MTR081RC : CONFIGURABLE_ROUT := (Actuate := 1, FeedbackType := 1, Feedback1 := 1, Feedback2 := 1, InputStatus := 1, OutputStatus := 1, FeedbackReactionTime := 250, O1 := 1, O2 := 1);   // Trimmer Scrap Conveyor FVNR Run Command
   FVNR_y778MTR080RC : CONFIGURABLE_ROUT := (Actuate := 1, FeedbackType := 1, Feedback1 := 1, Feedback2 := 1, InputStatus := 1, OutputStatus := 1, FeedbackReactionTime := 500, O1 := 1, O2 := 1);   // Shear Die Crank Motor FVNR Run Command
   FVR_y702MTR191_Flt : ALIAS FOR Flt_Starter.4;   // Rewind Pinch Roll Starter Fault ( 1= Fault)
   FVR_y702MTR191FC : CONFIGURABLE_ROUT := (FeedbackType := 1, InputStatus := 1, OutputStatus := 1, FeedbackReactionTime := 1000);   // Rewind Pinch Roll FVR Fwd Command
   FVR_y702MTR191RC : CONFIGURABLE_ROUT := (FeedbackType := 1, InputStatus := 1, OutputStatus := 1, FeedbackReactionTime := 1000);   // Rewind Pinch Roll FVR Rev Command
   FVR_y708MTR080_Flt : ALIAS FOR Flt_Starter.1;   // Flattener Drive Motor Starter Fault ( 1= Fault)
   FVR_y708MTR080FC : CONFIGURABLE_ROUT := (FeedbackType := 1, InputStatus := 1, OutputStatus := 1, FeedbackReactionTime := 250);   // Flattener Drive Motor FVR Fwd Command
   FVR_y708MTR080RC : CONFIGURABLE_ROUT := (FeedbackType := 1, InputStatus := 1, OutputStatus := 1, FeedbackReactionTime := 250);   // Flattener Drive Motor FVR Rev Command
   FVR_y708MTR250_Flt : ALIAS FOR Flt_Starter.0;   // Unwind Hold Down Roll Starter Fault ( 1= Fault)
   FVR_y708MTR250FC : CONFIGURABLE_ROUT := (FeedbackType := 1, InputStatus := 1, OutputStatus := 1, FeedbackReactionTime := 250);   // Unwind Hold Down Roll FVR Fwd Command
   FVR_y708MTR250RC : CONFIGURABLE_ROUT := (FeedbackType := 1, InputStatus := 1, OutputStatus := 1, FeedbackReactionTime := 250);   // Unwind Hold Down Roll FVR Rev Command
   FVR_y753MTR190_Flt : ALIAS FOR Flt_Starter.2;   // Trimmer Pinch Roll Starter Fault ( 1= Fault)
   FVR_y753MTR190FC : CONFIGURABLE_ROUT := (FeedbackType := 1, InputStatus := 1, OutputStatus := 1, FeedbackReactionTime := 250);   // Trimmer Pinch Roll FVR Fwd Command
   FVR_y753MTR190RC : CONFIGURABLE_ROUT := (FeedbackType := 1, InputStatus := 1, OutputStatus := 1, FeedbackReactionTime := 250);   // Trimmer Pinch Roll FVR Rev Command
   FVR_y761MTR081_Flt : ALIAS FOR Flt_Starter.3;   // Trimmer Scrap Conveyor Starter Fault ( 1= Fault)
   FVR_y778MTR080_Flt : ALIAS FOR Flt_Starter.5;   // Shear Die Crank Starter Fault ( 1= Fault)
   FVR_y802MTR080_Flt : ALIAS FOR Flt_Starter.6;   // Stacker Side Guide Lift Starter Fault ( 1= Fault)
   FVR_y802MTR080FC : CONFIGURABLE_ROUT := (FeedbackType := 1, InputStatus := 1, OutputStatus := 1, FeedbackReactionTime := 250);   // Stacker Side Guide Lift FVR Fwd Command
   FVR_y802MTR080RC : CONFIGURABLE_ROUT := (FeedbackType := 1, InputStatus := 1, OutputStatus := 1, FeedbackReactionTime := 250);   // Stacker Side Guide Lift FVR Rev Command
   FVR_y802MTR230_Flt : ALIAS FOR Flt_Starter.8;   // Scrap Horizontal Conveyor Starter Fault ( 1= Fault)
   FVR_y802MTR230FC : CONFIGURABLE_ROUT := (FeedbackType := 1, InputStatus := 1, OutputStatus := 1, FeedbackReactionTime := 250);   // Scrap Horizontal Conveyor FVR Fwd Command
   FVR_y802MTR230RC : CONFIGURABLE_ROUT := (FeedbackType := 1, InputStatus := 1, OutputStatus := 1, FeedbackReactionTime := 250);   // Scrap Horizontal Conveyor FVR Rev Command
   FVR_y802MTR231_Flt : ALIAS FOR Flt_Starter.7;   // Stacker Chain Conveyor Starter Fault ( 1= Fault)
   FVR_y802MTR231FC : CONFIGURABLE_ROUT := (FeedbackType := 1, InputStatus := 1, OutputStatus := 1, FeedbackReactionTime := 250);   // Stacker Chain Conveyor FVR Fwd Command
   FVR_y802MTR231RC : CONFIGURABLE_ROUT := (FeedbackType := 1, InputStatus := 1, OutputStatus := 1, FeedbackReactionTime := 250);   // Stacker Chain Conveyor FVR Rev Command
   G1_EstopRstCmd : BOOL;   // G1 Estop Reset Command ( 1= Reset Cmd)
   G1_FltRstCmd : BOOL;   // G1 Fault Reset Command ( 1= Reset Cmd)
   G1_IO : UDT_CardSts[32] := ([0].EntrySts := 16897, [0].Running := 1);   // G1 Point I/O
        [4]   // 1734-IE2C/C
   G1_IOSts_Flt : BOOL;   // G1 Point IO Module Fault ( 1= Faulted)
   G1_No_EStops : BOOL := 1;   // G1 No Estops ( 1= OK)
   G1_S11_ModFlt : ALIAS FOR Flt_Modules[0].15;   // G1 Point I/O Slot11 Module Fault (1 = Fault)
   G1_S12_ModFlt : ALIAS FOR Flt_Modules[0].16;   // G1 Point I/O Slot12 Module Fault (1 = Fault)
   G1_SolPwrEn : BOOL := 1;   // G1 Solenoid Safe-Off Enable ( 1= Enable )
   H1_EstopRstCmd : BOOL;   // H1 Estop Reset Command ( 1= Reset Cmd)
   H1_FltRstCmd : BOOL;   // H1 Fault Reset Command ( 1= Reset Cmd)
   H1_IO : UDT_CardSts[32] := ([0].EntrySts := 16897, [0].Running := 1);   // H1 Point I/O
        [4]   // 1734-IE2C/C
   H1_IOSts_Flt : BOOL;   // H1 Point IO Module Fault ( 1= Faulted)
   H1_No_EStops : BOOL := 1;   // H1 No Estops ( 1= OK)
   H1_S5_ModFlt : ALIAS FOR Flt_Modules[0].17;   // H1 Point I/O Slot05 Module Fault (1 = Fault)
   H1_S6_ModFlt : ALIAS FOR Flt_Modules[0].18;   // H1 Point I/O Slot06 Module Fault (1 = Fault)
   H1_SolPwrEn : BOOL := 1;   // H1 Solenoid Safe-Off Enable ( 1= Enable )
   HB_Citect : BOOL := 1;   // Heartbeat Citect Reflect
   HydPumps_AutoStart : BOOL;   // (From Mach) Hydraulic Pumps Auto Start Active
   IOCards_OK : DINT;   // Point I/O Cards OK
        .0   // MCC I/O Cards OK ( 1= OK)
        .1   // Op Stations (Entry Section) I/O Cards OK ( 1= OK)
        .2   // Op Stations (Exit Section) I/O Cards OK ( 1= OK)
        .3   // General I/O I/O Cards OK ( 1= OK)
        .4   // General I/O I/O Cards OK ( 1= OK)
        .31   // ALL I/O Cards OK ( 1= OK)
   jay : BOOL := 1;
   Line_CTC_CoastStop : BOOL;   // Line Coast Stop ( 1= Coast Stop) (Condition Exists)
   Line_CTL_CoastStop : BOOL;   // Line Coast Stop ( 1= Coast Stop) (Condition Exists)
   Line_No_Estop : DINT := -2147483645;   // Line Estop Summation ( 1= No Estop PB's) (Pressed)
   Line_NoP2P_CommFlts : BOOL := 1;   // Line No Peer to Peer Comm Faults ( 1= OK)
   Line_Total_CoastStop : BOOL;   // Line Coast Stop ( 1= Coast Stop) (Condition Exists)
   Line_TotalMode : BOOL := 1;   // Line TOTAL Mode ( 1= Total Mode) (0 = Coil to Coil)
   LineSts : UDT_SysStatus := (Heartbeat := 1, CoastStop_CTC := 1, CoastStop_CTL := 1, CoastStop_Total := 1, No_CTC_EStops := 1, No_CTL_EStops := 1, No_Total_Estops := 1, No_CTC_Faults := 1, No_CTL_Faults := 1, No_Total_Faults := 1, CTCStopTimer.PRE := 5000, CTLStopTimer.PRE := 5000, TotalStopTimer.PRE := 5000);
   Local_ModFlts : DINT := 514;   // Local Card Fault Status
        .1   // Slot 01
        .2   // Slot 02 1756-EN2T Card Fault ( 1= Fault)
        .3   // Slot 03 1756-EN2T Card Fault ( 1= Fault)
        .9   // Slot 09
        .16   // Slot 16 1756-EN2T Card Fault ( 1= Fault)
   Local_Networks_OK : BOOL := 1;   // Local Network CARDS OK ( 1= OK)
   Local_Slot : UDT_CardSts[17] := ([1].EntrySts := 24576, [2].EntrySts := 16897, [2].Running := 1, [3].EntrySts := 16897, [3].Running := 1, [4].EntrySts := 16897, [4].Running := 1, [5].EntrySts := 16897, [5].Running := 1, [6].EntrySts := 16897, [6].Running := 1, [7].EntrySts := 16897, [7].Running := 1, [9].EntrySts := 24576, [16].EntrySts := 16897, [16].Running := 1); {access Read Only}   // Safety Processor
        [8]   // 1756-L75 -
        [2]   // 1756-EN2T -
        [3]   // 1756-EN2T -
        [16]   // 1756-EN2T -
   LubePumps_AutoStart : BOOL;   // (From Mach) Lube Pumps Auto Start Active
   Machine_HB_Flt : BOOL;   // Machine Heartbeat Fault ( 1= Fault)
   Machine_HB_TOF : TIMER := (PRE := 1000);   // Machine Heartbeat Timer Off
   Machine_HB_TON : TIMER := (PRE := 1000, ACC := 100, EN := 1, TT := 1);   // Machine Heartbeat Timer On
   Map_Citect : DINT[5] := ([0] := 1);   // Mapped From Shear Citect System
        [0].0   // Citect Heartbeat Fault ( 1= Fault)
   Map_Mach : DINT[5] := ([0] := 4225);   // From Machine Processor
        [0].0   // (From Machine) Heartbeat Pulse
        [0].1   // Unwind Hold Down Roll Forward Command ( 1= Run Fwd )
        [0].2   // Unwind Hold Down Roll Reverse Command ( 1= Run Rev)
        [0].3   // Flattener Forward Command ( 1= Run Fwd )
        [0].4   // Flattener Reverse Command ( 1= Run Rev)
        [0].5   // Trimmer Pinch Roll Forward Command ( 1= Run Fwd )
        [0].6   // Trimmer Pinch Roll Reverse Command ( 1= Run Rev)
        [0].7   // Trimmer Scrap Conveyor Run Command ( 1= Run )
        [0].8   // Rewind Pinch Roll Forward Command ( 1= Run Fwd )
        [0].9   // Rewind Pinch Roll Reverse Command ( 1= Run Rev)
        [0].10   // Unwind Coil Car Safety Reset PB
        [0].11   // Line Emergency Stop Reset PBL
        [0].12   // Line TOTAL Mode ( 1= Total Mode) (0 = Coil to Coil)
   Map_ShDie : DINT[5] := ([0] := 3);   // Mapped From Shear Die Processor
        [0].1   // Shear Die Crank Run Command ( 1= Run)
        [0].2   // Scrap Horizontal Conveyor Fwd Cmd ( 1= Run Fwd)
        [0].3   // Scrap Horizontal Conveyor Rev Cmd ( 1= Run Rev)
        [0].4   // Stacker Chain Fwd Cmd
        [0].5   // Stacker Chain Rev Cmd
        [0].7   // Stacker Side Guide Lift Rev Cmd/Dwn
        [0].6   // Stacker Side Guide Lift Fwd Cmd/Up
        [0].8   // Shear Emergency Stop Reset PBL
        [0].0   // (From Shear Die) Heartbeat Pulse
        [0].9   // Line Emergency Stop Reset PBL
   MCC1_IO : UDT_CardSts[32] := ([0].EntrySts := 16897, [0].Running := 1);   // MCC1 Point I/O
        [13]   // 1734-IE2V/C
   MCC1_IOSts_Flt : BOOL;   // MCC1 Point IO Module Fault ( 1= Faulted)
   MCC1_S1_ModFlt : ALIAS FOR Flt_Modules[2].0;   // MCC1 Point I/O Slot01 Module Fault (1 = Fault)
   MCC1_S6_ModFlt : ALIAS FOR Flt_Modules[2].1;   // MCC1 Point I/O Slot06 Module Fault (1 = Fault)
   MCC2_IO : UDT_CardSts[32] := ([0].EntrySts := 28928);   // MCC2 Point I/O
        [13]   // 1734-IE2V/C
   MCC2_IOSts_Flt : BOOL;   // MCC2 Point IO Module Fault ( 1= Faulted)
   MCC2_S1_ModFlt : ALIAS FOR Flt_Modules[2].2;   // MCC2 Point I/O Slot01 Module Fault (1 = Fault)
   MCC2_S2_ModFlt : ALIAS FOR Flt_Modules[2].3;   // MCC2 Point I/O Slot02 Module Fault (1 = Fault)
   MCC3_IO : UDT_CardSts[32] := ([0].EntrySts := 16897, [0].Running := 1);   // MCC3 Point I/O
   MCC3_IOSts_Flt : BOOL;   // MCC3 Point IO Module Fault ( 1= Faulted)
   MCC3_S1_ModFlt : ALIAS FOR Flt_Modules[2].4;   // MCC3 Point I/O Slot01 Module Fault (1 = Fault)
   MCC3_S3_ModFlt : ALIAS FOR Flt_Modules[2].5;   // MCC3 Point I/O Slot03 Module Fault (1 = Fault)
   MCC3_S4_ModFlt : ALIAS FOR Flt_Modules[2].6;   // MCC3 Point I/O Slot04 Module Fault (1 = Fault)
   MCC4_IO : UDT_CardSts[32] := ([0].EntrySts := 16897, [0].Running := 1);   // MCC4 Point I/O
   MCC4_IOSts_Flt : BOOL;   // MCC-4 Point IO Module Fault ( 1= Faulted)
   MCC4_S1_ModFlt : ALIAS FOR Flt_Modules[2].7;   // MCC4 Point I/O Slot01 Module Fault (1 = Fault)
   MCC4_S3_ModFlt : ALIAS FOR Flt_Modules[2].8;   // MCC4 Point I/O Slot03 Module Fault (1 = Fault)
   MCC4_S4_ModFlt : ALIAS FOR Flt_Modules[2].9;   // MCC4 Point I/O Slot04 Module Fault (1 = Fault)
   MCC5_IO : UDT_CardSts[32] := ([0].EntrySts := 28928);   // MCC5 Point I/O
   MCC5_IOSts_Flt : BOOL;   // MCC-5 Point IO Module Fault ( 1= Faulted)
   MCC5_S1_ModFlt : ALIAS FOR Flt_Modules[2].10;   // MCC5 Point I/O Slot01 Module Fault (1 = Fault)
   MCC5_S3_ModFlt : ALIAS FOR Flt_Modules[2].11;   // MCC5 Point I/O Slot03 Module Fault (1 = Fault)
   MCC5_S4_ModFlt : ALIAS FOR Flt_Modules[2].12;   // MCC5 Point I/O Slot04 Module Fault (1 = Fault)
   MCC5_S5_ModFlt : ALIAS FOR Flt_Modules[2].13;   // MCC5 Point I/O Slot05 Module Fault (1 = Fault)
   OS11_EstopRstCmd : BOOL;   // OS11 Estop Reset Command ( 1= Reset Cmd)
   OS11_FltRstCmd : BOOL;   // OS11 Fault Reset Command ( 1= Reset Cmd)
   OS11_IO : UDT_CardSts[32] := ([0].EntrySts := 16897, [0].Running := 1);   // OS11 Point I/O
        [4]   // 1734-IE2C/C
   OS11_IOSts_Flt : BOOL;   // OS11 Point IO Module Fault ( 1= Faulted)
   OS11_No_EStops : BOOL := 1;   // OS11 No Estops ( 1= OK)
   OS11_S1_ModFlt : ALIAS FOR Flt_Modules[1].11;   // OS11 Point I/O Slot01 Module Fault (1 = Fault)
   OS13_EstopRstCmd : BOOL;   // OS13 Estop Reset Command ( 1= Reset Cmd)
   OS13_FltRstCmd : BOOL;   // OS13 Fault Reset Command ( 1= Reset Cmd)
   OS13_IO : UDT_CardSts[32] := ([0].EntrySts := 16897, [0].Running := 1);   // OS13 Point I/O
        [4]   // 1734-IE2C/C
   OS13_IOSts_Flt : BOOL;   // OS13 Point IO Module Fault ( 1= Faulted)
   OS13_No_EStops : BOOL := 1;   // OS13 No Estops ( 1= OK)
   OS13_S1_ModFlt : ALIAS FOR Flt_Modules[1].12;   // OS13 Point I/O Slot01 Module Fault (1 = Fault)
   OS14_EstopRstCmd : BOOL;   // OS14 Estop Reset Command ( 1= Reset Cmd)
   OS14_FltRstCmd : BOOL;   // OS14 Fault Reset Command ( 1= Reset Cmd)
   OS14_IO : UDT_CardSts[32] := ([0].EntrySts := 16897, [0].Running := 1);   // OS14 Point I/O
        [13]   // 1734-IE2V/C
   OS14_IOSts_Flt : BOOL;   // OS14 Point IO Module Fault ( 1= Faulted)
   OS14_No_EStops : BOOL := 1;   // OS14 No Estops ( 1= OK)
   OS14_S1_ModFlt : ALIAS FOR Flt_Modules[1].13;   // OS14 Point I/O Slot01 Module Fault (1 = Fault)
   OS14_Shear_EstopRstCmd : BOOL;   // OS14_Shear Estop Reset Command ( 1= Reset Cmd)
   OS14_Shear_FltRstCmd : BOOL;   // OS14_Shear Fault Reset Command ( 1= Reset Cmd)
   OS14_Shear_No_EStops : BOOL := 1;   // OS14_Shear No Estops ( 1= OK)
   OS15_EstopRstCmd : BOOL;   // OS15 Estop Reset Command ( 1= Reset Cmd)
   OS15_FltRstCmd : BOOL;   // OS15 Fault Reset Command ( 1= Reset Cmd)
   OS15_IO : UDT_CardSts[32] := ([0].EntrySts := 16897, [0].Running := 1);   // OS15 Point I/O
   OS15_IOSts_Flt : BOOL;   // OS15 Point IO Module Fault ( 1= Faulted)
   OS15_No_EStops : BOOL := 1;   // OS15 No Estops ( 1= OK)
   OS15_S1_ModFlt : ALIAS FOR Flt_Modules[1].14;   // OS15 Point I/O Slot01 Module Fault (1 = Fault)
   OS16_EstopRstCmd : BOOL;   // OS16 Estop Reset Command ( 1= Reset Cmd)
   OS16_FltRstCmd : BOOL;   // OS16 Fault Reset Command ( 1= Reset Cmd)
   OS16_IO : UDT_CardSts[32] := ([0].EntrySts := 16897, [0].Running := 1);   // OS16 Point I/O
   OS16_IOSts_Flt : BOOL;   // OS16 Point IO Module Fault ( 1= Faulted)
   OS16_No_EStops : BOOL := 1;   // OS16 No Estops ( 1= OK)
   OS16_S1_ModFlt : ALIAS FOR Flt_Modules[1].15;   // OS16 Point I/O Slot01 Module Fault (1 = Fault)
   OS1_EstopRstCmd : BOOL;   // OS1 Estop Reset Command ( 1= Reset Cmd)
   OS1_FltRstCmd : BOOL;   // OS1 Fault Reset Command ( 1= Reset Cmd)
   OS1_IO : UDT_CardSts[32] := ([0].EntrySts := 16897, [0].Running := 1);   // OS1 Point I/O
        [4]   // 1734-IE2C/C
   OS1_IOSts_Flt : BOOL;   // OS1 Point IO Module Fault ( 1= Faulted)
   OS1_No_EStops : BOOL := 1;   // OS1 No Estops ( 1= OK)
   OS1_S1_ModFlt : ALIAS FOR Flt_Modules[1].0;   // OS1 Point I/O Slot01 Module Fault (1 = Fault)
   OS2_EstopRstCmd : BOOL;   // OS2 Estop Reset Command ( 1= Reset Cmd)
   OS2_FltRstCmd : BOOL;   // OS2 Fault Reset Command ( 1= Reset Cmd)
   OS2_IO : UDT_CardSts[32] := ([0].EntrySts := 16897, [0].Running := 1, [1].EntrySts := 16897, [1].Running := 1, [3].EntrySts := 16899, [3].Running := 1, [4].EntrySts := 16897, [4].Running := 1, [5].EntrySts := 16897, [5].Running := 1, [6].EntrySts := 16897, [6].Running := 1, [7].EntrySts := 16897, [7].Running := 1); {access Read Only}   // OS2 Point I/O
   OS2_IOSts_Flt : BOOL;   // OS2 Point IO Module Fault ( 1= Faulted)
   OS2_No_EStops : BOOL := 1;   // OS2 No Estops ( 1= OK)
   OS2_S1_ModFlt : ALIAS FOR Flt_Modules[1].1;   // OS2 Point I/O Slot01 Module Fault (1 = Fault)
   OS3_EstopRstCmd : BOOL;   // OS3 Estop Reset Command ( 1= Reset Cmd)
   OS3_FltRstCmd : BOOL;   // OS3 Fault Reset Command ( 1= Reset Cmd)
   OS3_IO : UDT_CardSts[32] := ([0].EntrySts := 16897, [0].Running := 1);   // OS3 Point I/O
   OS3_IOSts_Flt : BOOL;   // OS3 Point IO Module Fault ( 1= Faulted)
   OS3_No_EStops : BOOL := 1;   // OS3 No Estops ( 1= OK)
   OS3_S1_ModFlt : ALIAS FOR Flt_Modules[1].2;   // OS3 Point I/O Slot01 Module Fault (1 = Fault)
   OS4_EstopRstCmd : BOOL;   // OS4 Estop Reset Command ( 1= Reset Cmd)
   OS4_FltRstCmd : BOOL;   // OS4 Fault Reset Command ( 1= Reset Cmd)
   OS4_No_EStops : BOOL := 1;   // OS4 No Estops ( 1= OK)
   OS4N_IO : UDT_CardSts[32] := ([0].EntrySts := 16897, [0].Running := 1);   // OS4N Point I/O
        [4]   // 1734-IE2C/C
   OS4N_IOSts_Flt : BOOL;   // OS4N Point IO Module Fault ( 1= Faulted)
   OS4N_S1_ModFlt : ALIAS FOR Flt_Modules[1].3;   // OS4N Point I/O Slot01 Module Fault (1 = Fault)
   OS4N_S5_ModFlt : ALIAS FOR Flt_Modules[1].4;   // OS4N Point I/O Slot05 Module Fault (1 = Fault)
   OS4N_SolPwrEn : BOOL := 1;   // OS4N Solenoid Safe-Off Enable ( 1= Enable )
   OS4S_IO : UDT_CardSts[32] := ([0].EntrySts := 16897, [0].Running := 1);   // OS4S Point I/O
        [4]   // 1734-IE2C/C
   OS4S_IOSts_Flt : BOOL;   // OS4S Point IO Module Fault ( 1= Faulted)
   OS4S_S1_ModFlt : ALIAS FOR Flt_Modules[1].5;   // OS4S Point I/O Slot01 Module Fault (1 = Fault)
   OS4S_S5_ModFlt : ALIAS FOR Flt_Modules[1].6;   // OS4S Point I/O Slot05 Module Fault (1 = Fault)
   OS4S_SolPwrEn : BOOL := 1;   // OS4S Solenoid Safe-Off Enable ( 1= Enable )
   OS5_EstopRstCmd : BOOL;   // OS5 Estop Reset Command ( 1= Reset Cmd)
   OS5_FltRstCmd : BOOL;   // OS5 Fault Reset Command ( 1= Reset Cmd)
   OS5_IO : UDT_CardSts[32] := ([0].EntrySts := 16897, [0].Running := 1);   // OS5 Point I/O
        [4]   // 1734-IE2C/C
   OS5_IOSts_Flt : BOOL;   // OS5 Point IO Module Fault ( 1= Faulted)
   OS5_No_EStops : BOOL := 1;   // OS5 No Estops ( 1= OK)
   OS5_S1_ModFlt : ALIAS FOR Flt_Modules[1].7;   // OS5 Point I/O Slot01 Module Fault (1 = Fault)
   OS6_EstopRstCmd : BOOL;   // OS6 Estop Reset Command ( 1= Reset Cmd)
   OS6_FltRstCmd : BOOL;   // OS6 Fault Reset Command ( 1= Reset Cmd)
   OS6_IO : UDT_CardSts[32] := ([0].EntrySts := 16897, [0].Running := 1);   // OS6 Point I/O
        [4]   // 1734-IE2C/C
   OS6_IOSts_Flt : BOOL;   // OS6 Point IO Module Fault ( 1= Faulted)
   OS6_No_EStops : BOOL := 1;   // OS6 No Estops ( 1= OK)
   OS6_S1_ModFlt : ALIAS FOR Flt_Modules[1].8;   // OS6 Point I/O Slot01 Module Fault (1 = Fault)
   OS8_EstopRstCmd : BOOL;   // OS8 Estop Reset Command ( 1= Reset Cmd)
   OS8_FltRstCmd : BOOL;   // OS8 Fault Reset Command ( 1= Reset Cmd)
   OS8_IO : UDT_CardSts[32] := ([0].EntrySts := 16897, [0].Running := 1);   // OS8 Point I/O
        [4]   // 1734-IE2C/C
   OS8_IOSts_Flt : BOOL;   // OS8 Point IO Module Fault ( 1= Faulted)
   OS8_No_EStops : BOOL := 1;   // OS8 No Estops ( 1= OK)
   OS8_S1_ModFlt : ALIAS FOR Flt_Modules[1].9;   // OS8 Point I/O Slot01 Module Fault (1 = Fault)
   OS9_EstopRstCmd : BOOL;   // OS9 Estop Reset Command ( 1= Reset Cmd)
   OS9_FltRstCmd : BOOL;   // OS9 Fault Reset Command ( 1= Reset Cmd)
   OS9_IO : UDT_CardSts[32] := ([0].EntrySts := 16897, [0].Running := 1);   // OS9 Point I/O
        [4]   // 1734-IE2C/C
   OS9_IOSts_Flt : BOOL;   // OS9 Point IO Module Fault ( 1= Faulted)
   OS9_No_EStops : BOOL := 1;   // OS9 No Estops ( 1= OK)
   OS9_S1_ModFlt : ALIAS FOR Flt_Modules[1].10;   // OS9 Point I/O Slot01 Module Fault (1 = Fault)
   Peer_Networks_OK : BOOL := 1;   // Peer Network CARDS OK ( 1= OK)
   PrCon_DrvsOff : BOOL;   // Product Conveyors (1-3) Drives OFF ( 1= OFF)
   PrCon_SafeTrqEn : BOOL := 1;   // Product Conveyors Safe-Trq Off Enable ( 1= Enable )
   PW_DrvsOff : BOOL;   // Paper Winder Drives OFF ( 1= OFF)
   PW_SafeTrqEn : BOOL := 1;   // Paper Winder Safe-Trq Off Enable ( 1= Enable )
   Rem_ModFlts : DINT;   // Remote IO Comm Faults
        .0   // A1 Point IO Comm Fault ( 1= Fault)
        .1   // C1 Point IO Comm Fault ( 1= Fault)
        .2   // CHPLC Point IO Comm Fault ( 1= Fault)
        .3   // D1 Point IO Comm Fault ( 1= Fault)
        .4   // DPD Point IO Comm Fault ( 1= Fault)
        .5   // E1 Point IO Comm Fault ( 1= Fault)
        .6   // F1 Point IO Comm Fault ( 1= Fault)
        .7   // G1 Point IO Comm Fault ( 1= Fault)
        .8   // MCC1 Point IO Comm Fault ( 1= Fault)
        .9   // MCC3 Point IO Comm Fault ( 1= Fault)
        .10   // OS11 Point IO Comm Fault ( 1= Fault)
        .11   // OS13 Point IO Comm Fault ( 1= Fault)
        .12   // OS1 Point IO Comm Fault ( 1= Fault)
        .13   // OS2 Point IO Comm Fault ( 1= Fault)
        .14   // OS3 Point IO Comm Fault ( 1= Fault)
        .15   // OS4N Point IO Comm Fault ( 1= Fault)
        .16   // OS4S Point IO Comm Fault ( 1= Fault)
        .17   // OS5 Point IO Comm Fault ( 1= Fault)
        .18   // OS6 Point IO Comm Fault ( 1= Fault)
        .19   // OS8 Point IO Comm Fault ( 1= Fault)
        .20   // OS9 Point IO Comm Fault ( 1= Fault)
        .21   // VS2 Point IO Comm Fault ( 1= Fault)
        .22   // MCC2 Point IO Comm Fault ( 1= Fault)
        .23   // SDPLC Point IO Comm Fault ( 1= Fault)
        .25   // MCC5 Point IO Comm Fault ( 1= Fault)
        .26   // OS16 Point IO Comm Fault ( 1= Fault)
        .27   // OS14 Point IO Comm Fault ( 1= Fault)
        .28   // H1 Point IO Comm Fault ( 1= Fault)
        .29   // OS15 Point IO Comm Fault ( 1= Fault)
        .24   // MCC4 Point IO Comm Fault ( 1= Fault)
   Rew_DrvsOff : BOOL;   // Rewind Drives OFF ( 1= OFF)
   REW_SafeOffEn : BOOL := 1;   // Rewind Safe-Off Enable ( 1= Enable )
   REW_SafeOffFltRst : BOOL;   // Rewind Safe-Off Fault Reset ( 1= Reset Cmd )
   RewPR_FVR_En : BOOL := 1;   // Rewind Pinch Roll FVR Enable ( 1= Enable )
   RewPR_FVR_FltRst : BOOL;   // Rewind Pinch Roll Fault Reset ( 1= Reset Cmd )
   RewPR_FVR_FwdCmd : BOOL;   // Rewind Pinch Roll Forward Command ( 1= Run Fwd )
   RewPR_FVR_RevCmd : BOOL;   // Rewind Pinch Roll Reverse Command ( 1= Run Rev)
   Rodney_Always : BOOL;
   Rodney_True : BOOL := 1;
   SafeOff_y172CR460 : CONFIGURABLE_ROUT := (Actuate := 1, FeedbackType := 1, Feedback1 := 1, Feedback2 := 1, InputStatus := 1, OutputStatus := 1, FeedbackReactionTime := 250, O1 := 1, O2 := 1);   // Shear Die Main Contactor Relay
   SafeOff_y172CR460_Flt : ALIAS FOR Flt_SafeOff[0].0;   // Shear Die Main Contactor Relay Fault ( 1= Fault)
   SafeOff_y172CR510 : CONFIGURABLE_ROUT := (Actuate := 1, FeedbackType := 1, Feedback1 := 1, Feedback2 := 1, InputStatus := 1, OutputStatus := 1, FeedbackReactionTime := 250, O1 := 1, O2 := 1);   // Shear Die Drive Enable Relay
   SafeOff_y172CR510_Flt : ALIAS FOR Flt_SafeOff[0].1;   // Shear Die Drive Enable Relay Fault ( 1= Fault)
   SafeOff_y613CR460 : CONFIGURABLE_ROUT := (Actuate := 1, FeedbackType := 1, Feedback1 := 1, Feedback2 := 1, InputStatus := 1, OutputStatus := 1, FeedbackReactionTime := 250, O1 := 1, O2 := 1);   // Unwind Op Side Main Contactor Relay
   SafeOff_y613CR460_Flt : ALIAS FOR Flt_SafeOff[0].2;   // Unwind Op Side Main Contactor Relay Fault ( 1= Fault)
   SafeOff_y613CR510 : CONFIGURABLE_ROUT := (Actuate := 1, FeedbackType := 1, Feedback1 := 1, Feedback2 := 1, InputStatus := 1, OutputStatus := 1, FeedbackReactionTime := 250, O1 := 1, O2 := 1);   // Unwind Op Side Drive Enable Relay
   SafeOff_y613CR510_Flt : ALIAS FOR Flt_SafeOff[0].3;   // Unwind Op Side Drive Enable Relay Fault ( 1= Fault)
   SafeOff_y613CR550 : CONFIGURABLE_ROUT := (Actuate := 1, FeedbackType := 1, Feedback1 := 1, Feedback2 := 1, InputStatus := 1, OutputStatus := 1, FeedbackReactionTime := 250, O1 := 1, O2 := 1);   // Unwind Drive Side Main Contactor Relay
   SafeOff_y613CR550_Flt : ALIAS FOR Flt_SafeOff[0].4;   // Unwind Drive Side Main Contactor Relay Fault ( 1= Fault)
   SafeOff_y613CR590 : CONFIGURABLE_ROUT := (Actuate := 1, FeedbackType := 1, Feedback1 := 1, Feedback2 := 1, InputStatus := 1, OutputStatus := 1, FeedbackReactionTime := 250, O1 := 1, O2 := 1);   // Unwind Drive Side Drive Enable Relay
   SafeOff_y613CR590_Flt : ALIAS FOR Flt_SafeOff[0].5;   // Unwind Drive Side Drive Enable Relay Fault ( 1= Fault)
   SafeOff_y613CR630 : CONFIGURABLE_ROUT := (Actuate := 1, FeedbackType := 1, Feedback1 := 1, Feedback2 := 1, InputStatus := 1, OutputStatus := 1, FeedbackReactionTime := 250, O1 := 1, O2 := 1);   // #1 Entry Bridle Roll 2 Main Contactor Relay
   SafeOff_y613CR630_Flt : ALIAS FOR Flt_SafeOff[0].6;   // #1 Entry Bridle Roll 2 Main Contactor Relay Fault ( 1= Fault)
   SafeOff_y613CR670 : CONFIGURABLE_ROUT := (Actuate := 1, FeedbackType := 1, Feedback1 := 1, Feedback2 := 1, InputStatus := 1, OutputStatus := 1, FeedbackReactionTime := 250, O1 := 1, O2 := 1);   // #1 Entry Bridle Roll 2 Drive Enable Relay
   SafeOff_y613CR670_Flt : ALIAS FOR Flt_SafeOff[0].7;   // #1 Entry Bridle Roll 2 Drive Enable Relay Fault ( 1= Fault)
   SafeOff_y613CR710 : CONFIGURABLE_ROUT := (Actuate := 1, FeedbackType := 1, Feedback1 := 1, Feedback2 := 1, InputStatus := 1, OutputStatus := 1, FeedbackReactionTime := 250, O1 := 1, O2 := 1);   // #2 Entry Bridle Roll 3 Main Contactor Relay
   SafeOff_y613CR710_Flt : ALIAS FOR Flt_SafeOff[0].8;   // #2 Entry Bridle Roll 3 Main Contactor Relay Fault ( 1= Fault)
   SafeOff_y613CR750 : CONFIGURABLE_ROUT := (Actuate := 1, FeedbackType := 1, Feedback1 := 1, Feedback2 := 1, InputStatus := 1, OutputStatus := 1, FeedbackReactionTime := 250, O1 := 1, O2 := 1);   // #2 Entry Bridle Roll 3 Drive Enable Relay
   SafeOff_y613CR750_Flt : ALIAS FOR Flt_SafeOff[0].9;   // #2 Entry Bridle Roll 3 Drive Enable Relay Fault ( 1= Fault)
   SafeOff_y614CR040 : CONFIGURABLE_ROUT := (Actuate := 1, FeedbackType := 1, Feedback1 := 1, Feedback2 := 1, InputStatus := 1, OutputStatus := 1, FeedbackReactionTime := 250, O1 := 1, O2 := 1);   // #1 Exit Bridle Roll 6 Main Contactor Relay
   SafeOff_y614CR040_Flt : ALIAS FOR Flt_SafeOff[0].10;   // #1 Exit Bridle Roll 6 Main Contactor Relay Fault ( 1= Fault)
   SafeOff_y614CR090 : CONFIGURABLE_ROUT := (Actuate := 1, FeedbackType := 1, Feedback1 := 1, Feedback2 := 1, InputStatus := 1, OutputStatus := 1, FeedbackReactionTime := 250, O1 := 1, O2 := 1);   // #1 Exit Bridle Roll 6 Drive Enable Relay
   SafeOff_y614CR090_Flt : ALIAS FOR Flt_SafeOff[0].11;   // #1 Exit Bridle Roll 6 Drive Enable Relay Fault ( 1= Fault)
   SafeOff_y614CR130 : CONFIGURABLE_ROUT := (Actuate := 1, FeedbackType := 1, Feedback1 := 1, Feedback2 := 1, InputStatus := 1, OutputStatus := 1, FeedbackReactionTime := 250, O1 := 1, O2 := 1);   // #2 Exit Bridle Roll 7 Main Contactor Relay
   SafeOff_y614CR130_Flt : ALIAS FOR Flt_SafeOff[0].12;   // #2 Exit Bridle Roll 7 Main Contactor Relay Fault ( 1= Fault)
   SafeOff_y614CR170 : CONFIGURABLE_ROUT := (Actuate := 1, FeedbackType := 1, Feedback1 := 1, Feedback2 := 1, InputStatus := 1, OutputStatus := 1, FeedbackReactionTime := 250, O1 := 1, O2 := 1);   // #2 Exit Bridle Roll 7 Drive Enable Relay
   SafeOff_y614CR170_Flt : ALIAS FOR Flt_SafeOff[0].13;   // #2 Exit Bridle Roll 7 Drive Enable Relay Fault ( 1= Fault)
   SafeOff_y614CR210 : CONFIGURABLE_ROUT := (Actuate := 1, FeedbackType := 1, Feedback1 := 1, Feedback2 := 1, InputStatus := 1, OutputStatus := 1, FeedbackReactionTime := 250, O1 := 1, O2 := 1);   // Rewind Main Contactor Relay
   SafeOff_y614CR210_Flt : ALIAS FOR Flt_SafeOff[0].14;   // Rewind Main Contactor Relay Fault ( 1= Fault)
   SafeOff_y614CR250 : CONFIGURABLE_ROUT := (Actuate := 1, FeedbackType := 1, Feedback1 := 1, Feedback2 := 1, InputStatus := 1, OutputStatus := 1, FeedbackReactionTime := 250, O1 := 1, O2 := 1);   // Rewind Drive Enable Relay
   SafeOff_y614CR250_Flt : ALIAS FOR Flt_SafeOff[0].15;   // Rewind Drive Enable Relay Fault ( 1= Fault)
   Safety_HB_TOF : TIMER := (PRE := 250, ACC := 50, EN := 1, TT := 1);   // Safety Heartbeat Pulse Time Off
   Safety_HB_TON : TIMER := (PRE := 250);   // Safety Heartbeat Pulse Time On
   SC_DrvsOff : BOOL;   // Scrap Chop Conveyor Drives OFF ( 1= OFF)
   SC_SafeTrqEn : BOOL := 1;   // Scrap Chopper Safe-Trq Off Enable ( 1= Enable )
   ScHorCon_FVR_En : BOOL := 1;   // Scrap Horizontal Conveyor FVR Enable ( 1= Enable )
   ScHorCon_FVR_FltRst : BOOL;   // Scrap Horizontal Conveyor Fault Reset ( 1= Reset Cmd )
   ScHorCon_FVR_FwdCmd : BOOL;   // Scrap Horizontal Conveyor Forward Command ( 1= Run Fwd )
   ScHorCon_FVR_RevCmd : BOOL;   // Scrap Horizontal Conveyor Reverse Command ( 1= Run Rev)
   ScInCon_DrvsOff : BOOL;   // Scrap Incline Conveyor Drives OFF ( 1= OFF)
   ScInCon_SafeTrqEn : BOOL := 1;   // Scrap Incline Conveyor Safe-Trq Off Enable ( 1= Enable )
   ScrapModeOn : BOOL;   // Scrap Mode Selected ( 1= Requested)
   SDPLC_IO : UDT_CardSts[32] := ([0].EntrySts := 16897, [0].Running := 1, [1].EntrySts := 16897, [1].Running := 1, [3].EntrySts := 16899, [3].Running := 1, [4].EntrySts := 16897, [4].Running := 1, [5].EntrySts := 16897, [5].Running := 1, [6].EntrySts := 16897, [6].Running := 1, [7].EntrySts := 16897, [7].Running := 1); {access Read Only}   // SDPLC Point I/O
   SDPLC_IOSts_Flt : BOOL;   // SDPLC Point IO Module Fault ( 1= Faulted)
   SDPLC_S1_ModFlt : ALIAS FOR Flt_Modules[0].19;   // SDPLC Point I/O Slot01 Module Fault (1 = Fault)
   SDPLC_S2_ModFlt : ALIAS FOR Flt_Modules[0].20;   // SDPLC Point I/O Slot02 Module Fault (1 = Fault)
   SDPLC_SolPwrEn : BOOL := 1;   // SDPLC Solenoid Safe-Off Enable ( 1= Enable )
   Sfty_InstrFlts : DINT := 21511;   // Line Instruction Fault Word
        .0   // Estop Safety Instructions OK ( 1= No Faults)
        .1   // Safe-Off Safety Instructions OK ( 1= No Faults)
        .2   // FVR/FVNR Starters Safety Instructions OK ( 1= No Faults)
   Sfty_InstrFlts0_CTC : BOOL := 1;   // Coil To Coil Estop Safety Instructions OK ( 1= No Faults)
   Sfty_InstrFlts0_CTL : BOOL := 1;   // Cut To Length Estop Safety Instructions OK ( 1= No Faults)
   Sfty_InstrFlts0_Total : BOOL := 1;   // Total Mode Estop Safety Instructions OK ( 1= No Faults)
   Sfty_InstrFlts1_CTC : BOOL := 1;   // Coil To Coil Safe-Off Safety Instructions OK ( 1= No Faults)
   Sfty_InstrFlts1_CTL : BOOL := 1;   // Cut To Length Safe-Off Safety Instructions OK ( 1= No Faults)
   Sfty_InstrFlts1_Total : BOOL := 1;   // Total Mode Safe-Off Safety Instructions OK ( 1= No Faults)
   Sfty_InstrFlts2_CTC : BOOL := 1;   // Coil To Coil FVR/FVNR Starters Safety Instructions OK ( 1= No Faults)
   Sfty_InstrFlts2_CTL : BOOL := 1;   // Cut To Length FVR/FVNR Starters Safety Instructions OK ( 1= No Faults)
   Sfty_InstrFlts2_Total : BOOL := 1;   // Total Mode FVR/FVNR Starters Safety Instructions OK ( 1= No Faults)
   Sfty_ModFlts : DINT := 8199;   // Line Safety Module Fault Word
        .0   // General I/O Safety Module Faults ( 1= OK)
        .1   // Operator Station Safety Module Faults ( 1= OK)
        .2   // MCC Safety Module Faults ( 1= OK)
   Sfty_ModFlts0_CTC : BOOL := 1;   // Coil To Coil General I/O Safety Module Faults ( 1= OK)
   Sfty_ModFlts0_CTL : BOOL := 1;   // Cut To Length General I/O Safety Module Faults ( 1= OK)
   Sfty_ModFlts0_Total : BOOL := 1;   // Total Mode General I/O Safety Module Faults ( 1= OK)
   Sfty_ModFlts1_CTC : BOOL := 1;   // Coil To Coil Operator Station Safety Module Faults ( 1= OK)
   Sfty_ModFlts1_CTL : BOOL := 1;   // Cut To Length Operator Station Safety Module Faults ( 1= OK)
   Sfty_ModFlts1_Total : BOOL := 1;   // Total Mode Operator Station Safety Module Faults ( 1= OK)
   Sfty_ModFlts2_CTC : BOOL := 1;   // Coil To Coil MCC Safety Module Faults ( 1= OK)
   Sfty_ModFlts2_CTL : BOOL := 1;   // Cut To Lenght MCC Safety Module Faults ( 1= OK)
   Sfty_ModFlts2_Total : BOOL := 1;   // Total Mode MCC Safety Module Faults ( 1= OK)
   SftyMap_Citect : DINT[5] := ([0] := 1);   // SAFETY MAPPED From Citect System
        [0].0   // (SAFETY MAPPED) Citect System Comm Fault ( 1= Fault)
   SftyMap_Mach : DINT[5] := ([0] := 4225);   // SAFETY MAPPED From Machine Processor
        [0].0   // (SAFETY MAPPED) (From Machine) Heartbeat Pulse
        [0].9   // (SAFETY MAPPED) Rewind Pinch Roll Reverse Command ( 1= Run Rev)
        [0].10   // (SAFETY MAPPED) Unwind Coil Car Safety Reset PB
        [0].8   // (SAFETY MAPPED) Pinch Roll Forward Command ( 1= Run Fwd )
        [0].6   // (SAFETY MAPPED) Trimmer Pinch Roll Reverse Command ( 1= Run Rev)
        [0].7   // (SAFETY MAPPED) Trimmer Scrap Conveyor Run Command ( 1= Run )
        [0].4   // (SAFETY MAPPED) Flattener Reverse Command ( 1= Run Rev)
        [0].2   // (SAFETY MAPPED) Unwind Hold Down Roll Reverse Command ( 1= Run Rev)
        [0].3   // (SAFETY MAPPED) Flattener Forward Command ( 1= Run Fwd )
        [0].1   // (SAFETY MAPPED) Unwind Hold Down Roll Forward Command ( 1= Run Fwd )
        [0].5   // (SAFETY MAPPED) Trimmer Pinch Roll Forward Command ( 1= Run Fwd )
        [0].11   // SAFETY MAPPED Line Emergency Stop Reset PBL
        [0].12   // (SAFTY MAPPED) Line TOTAL Mode ( 1= Total Mode) (0 = Coil to Coil)
   SftyMap_ShDie : DINT[5] := ([0] := 3);   // SAFETY MAPPED From Shear Die Processor
        [0].7   // (SAFETY MAPPED) Stacker Side Guide Lift Rev Cmd/Dwn
        [0].3   // (SAFETY MAPPED) Scrap Horizontal Conveyor Rev Cmd ( 1= Run Rev)
        [0].0   // (SAFETY MAPPED) (From Shear Die) Heartbeat Pulse
        [0].1   // (SAFETY MAPPED) Shear Die Crank Run Command ( 1= Run)
        [0].2   // (SAFETY MAPPED) Scrap Horizontal Conveyor Rev Cmd ( 1= Run Rev)
        [0].4   // (SAFETY MAPPED) Stacker Chain Fwd Cmd
        [0].6   // (SAFETY MAPPED) Stacker Side Guide Lift Fwd Cmd/Up
        [0].5   // (SAFETY MAPPED) Stacker Chain Rev Cmd
        [0].8   // SAFETY MAPPED Shear Emergency Stop Reset PBL
        [0].9   // SAFETY MAPPED Line Emergency Stop Reset PBL
   SGWA_DrvsOff : BOOL;   // Side Guide Width Adjust Drives OFF ( 1= OFF)
   SGWA_SafeTrqEn : BOOL := 1;   // Side Guide Width Adjust Safe-Trq Off Enable ( 1= Enable )
   Shear_CoastStop : BOOL;   // Shear Coast Stop ( 1= Coast Stop) (Condition Exists)
   Shear_HB_Flt : BOOL;   // Shear Heartbeat Fault ( 1= Fault)
   Shear_HB_TOF : TIMER := (PRE := 1200);   // Shear Heartbeat Pulse Time Off
   Shear_HB_TON : TIMER := (PRE := 1200, EN := 1, TT := 1);   // Shear Heartbeat Pulse Time On
   ShearSts : UDT_ShearStatus := (CoastStop := 1, No_EStops := 1, No_Faults := 1);
   SkBkSt_DrvsOff : BOOL;   // Stacker Backstop Drives OFF ( 1= OFF)
   SkBkSt_SafeTrqEn : BOOL := 1;   // Stacker Back Stop Safe-Trq Off Enable ( 1= Enable )
   SkBlwr_DrvsOff : BOOL;   // Stacker Blower Drives OFF ( 1= OFF)
   SkBlwr_SafeTrqEn : BOOL := 1;   // Stacker Blower Safe-Trq Off Enable ( 1= Enable )
   SkChain_FVR_En : BOOL := 1;   // Stacker Chain FVR Enable ( 1= Enable )
   SkChain_FVR_FltRst : BOOL;   // Stacker Chain Fault Reset ( 1= Reset Cmd )
   SkChain_FVR_FwdCmd : BOOL;   // Stacker Chain Forward Command ( 1= Run Fwd )
   SkChain_FVR_RevCmd : BOOL;   // Stacker Chain Reverse Command ( 1= Run Rev)
   SkSGLift_FVR_En : BOOL := 1;   // Stacker Side Guide Lift FVR Enable ( 1= Enable )
   SkSGLift_FVR_FltRst : BOOL;   // Stacker Side Guide Lift Fault Reset ( 1= Reset Cmd )
   SkSGLift_FVR_FwdCmd : BOOL;   // Stacker Side Guide Lift Forward Command ( 1= Run Fwd )
   SkSGLift_FVR_RevCmd : BOOL;   // Stacker Side Guide Lift Reverse Command ( 1= Run Rev)
   Sr_DrvsOff : BOOL;   // Shear Pinch Roll/ Metering Back Up Drives OFF ( 1= OFF)
   Sr_SafeTrqEn : BOOL := 1;   // Shear Pinch Roll/ Back Up Roll Safe-Trq Off Enable ( 1= Enable )
   SrCon_DrvsOff : BOOL;   // Shear Conveyor Drives OFF ( 1= OFF)
   SrCon_SafeTrqEn : BOOL := 1;   // Shear Conveyor Safe-Trq Off Enable ( 1= Enable )
   SrDie_DrvsOff : BOOL;   // Shear Die Drives OFF ( 1= OFF)
   SrDie_SafeOffEn : BOOL := 1;   // Shear Die Safe-Off Enable ( 1= Enable )
   SrDie_SafeOffFltRst : BOOL;   // Shear Die Safe-Off Fault Reset ( 1= Reset Cmd )
   SrDieCrnk_FVNR_En : BOOL := 1;   // Shear Die Crank FVNR Enable ( 1= Enable )
   SrDieCrnk_FVNR_FltRst : BOOL;   // Shear Die Crank FVNR Enable ( 1= Enable )
   SrDieCrnk_FVNR_RunCmd : BOOL := 1;   // Shear Die Crank Run Command ( 1= Run )
   SrPRLubePump_AutoStart : BOOL;   // (From Mach) Shear Pinch Roll Lube Pump Auto Start Command
   StHydPump_AutoStart : BOOL;   // (From Mach) Sheeter Hydraulic Pump Auto Start Command
   StPR_DrvsOff : BOOL;   // Sheeter Pinch Roll Drives OFF ( 1= OFF)
   StPR_SafeTrqEn : BOOL := 1;   // Sheeter Pinch Roll Safe-Trq Off Enable ( 1= Enable )
   StPRLubePump_AutoStart : BOOL;   // (From Mach) Sheeter Pinch Roll Lube Pump Auto Start Command
   Sy_ClrFlt : BOOL;   // System Clear Fault
   Test_RN : BOOL := 1;
   TK_DrvsOff : BOOL;   // Trimmer Knives/ Width Adjust Drives OFF ( 1= OFF)
   TK_SafeTrqEn : BOOL := 1;   // Trimmer Knife Safe-Trq Off Enable ( 1= Enable )
   ToCitect : DINT[64] := ([0] := 1048574, [1] := 14, [2] := 14);   // (To Citect)
        [0].30   // (To Citect)
        [0].21   // (To Citect)
        [0].20   // (To Citect)
        [0].22   // (To Citect)
        [0].23   // (To Citect)
        [0].24   // (To Citect)
        [0].25   // (To Citect)
        [0].26   // (To Citect)
        [0].27   // (To Citect)
        [0].28   // (To Citect)
        [0].29   // (To Citect)
        [0].1   // (To Citect) OS1 Line EStop Pushbutton
        [0].2   // (To Citect) OS2 Line EStop Pushbutton
        [0].31   // (To Citect)
        [0].4   // (To Citect) OS4N Line EStop Pushbutton
        [1]   // (To Citect)
        [0].13   // (To Citect) OS14 Shear Estop Pushbutton
        [0].18   // (To Citect) G1 Tripwire Line EStop
        [0].3   // (To Citect) OS3 Line EStop Pushbutton
        [0].5   // (To Citect) OS4S Line EStop Pushbutton
        [0].6   // (To Citect) OS5 Line EStop Pushbutton
        [0].7   // (To Citect) OS6 Line EStop Pushbutton
        [0].8   // (To Citect) OS8 Line EStop Pushbutton
        [0].9   // (To Citect) OS9 Line EStop Pushbutton
        [0].10   // (To Citect) OS11 Line EStop Pushbutton
        [0].11   // (To Citect) OS13 Line EStop Pushbutton
        [0].12   // (To Citect) OS14 Line EStop Pushbutton
        [0].14   // (To Citect) OS15 Line EStop Pushbutton
        [0].15   // (To Citect) OS16 Line EStop Pushbutton
        [0].16   // (To Citect) DPD Line EStop Pushbutton
        [0].17   // (To Citect) DPD (In Pit) Line EStop Pushbutton
        [0].19   // (To Citect) H1 Line EStop Pushbutton
        [0].0   // (To Citect) Heartbeat
        [1].1   // (From Safety) Line Safety Status Coast Stop ( 0 = Coast Stop) ( 1= OK)
        [1].2   // (From Safety) Line Safety Status EStop ( 0 = EStop) ( 1= OK)
        [1].3   // (From Safety) Line Safety Status No Faults ( 0 = Faults) ( 1= OK)
        [1].5   // (From Safety) Line Safety Status All Drives Off ( 1= All Off)
        [1].6   // (From Safety) Line Safety Status Safety Pwr On ( 1= All On)
        [2].1   // (From Safety) Shear Safety Status Coast Stop ( 0 = Coast Stop) ( 1= OK)
        [2].2   // (From Safety) Shear Safety Status EStop ( 0 = EStop) ( 1= OK)
        [2].5   // (From Safety) Shear Safety Status All Drives Off ( 1= All Off)
        [2].3   // (From Safety) Shear Safety Status No Faults ( 0 = Faults) ( 1= OK)
        [2].6   // (From Safety) Shear Safety Status Safety Pwr On ( 1= All On)
   ToCitect4 : DINT[64];   // (To Citect4)
        [0].0   // A1:O.Data[20].0 y406CR050 Line Solenoid Safe Off
        [0].1   // A1:O.Data[20].1 y406CR090 Coil Car Solenoid Safe Off
        [0].3   // A1:O.Data[20].3 y406CR170 Spare
        [0].2   // A1:O.Data[20].2 y406CR120 Spare
        [0].4   // A1:O.Data[20].4 A1_S20_4 (SPARE)
        [0].5   // A1:O.Data[20].5 A1_S20_5 (SPARE)
        [0].6   // A1:O.Data[20].6 A1_S20_6 (SPARE)
        [0].9   // A1:I.Data[21].1 x406LCB052 North/South Light Curtain Output B
        [0].8   // A1:I.Data[21].0 x406LCA047 North/South Light Curtain Output A
        [0].7   // A1:O.Data[20].7 A1_S20_7 (SPARE)
        [0].10   // A1:I.Data[21].2 A1_S21_2 (SPARE)
        [0].11   // A1:I.Data[21].3 A1_S21_3 (SPARE)
        [0].12   // A1:I.Data[21].4 A1_S21_4 (SPARE)
        [0].13   // A1:I.Data[21].5 A1_S21_5 (SPARE)
        [0].14   // A1:I.Data[21].6 A1_S21_6 (SPARE)
        [0].15   // A1:I.Data[21].7 A1_S21_7 (SPARE)
        [0].16   // C1:O.Data[12].0 y435CR050 Solenoid Safe Off
        [0].17   // C1:O.Data[12].1 C1_S12_1 (SPARE)
        [0].18   // C1:O.Data[12].2 C1_S12_2 (SPARE)
        [0].19   // C1:O.Data[12].3 C1_S12_3 (SPARE)
        [0].20   // C1:O.Data[12].4 C1_S12_4 (SPARE)
        [0].21   // C1:O.Data[12].5 C1_S12_5 (SPARE)
        [0].22   // C1:O.Data[12].6 C1_S12_6 (SPARE)
        [0].23   // C1:O.Data[12].7 C1_S12_7 (SPARE)
        [0].24   // CHPLC:I.Data[1].0 x613CR460 Unwind Operator Side Main Contactor Safety Relay
        [0].25   // CHPLC:I.Data[1].1 x613CR510 Unwind Operator Side Drive Enable Safety Relay
        [0].26   // CHPLC:I.Data[1].2 x613CR550 Unwind Drive Side Main Contactor Safety Relay
        [0].27   // CHPLC:I.Data[1].3 x613CR590 Unwind Drive Side Drive Enable Safety Relay
        [0].28   // CHPLC:I.Data[1].4 x613CR630 #1 Entry Bridle Roll 2 Main Contactor Safety Relay
        [0].29   // CHPLC:I.Data[1].5 x613CR670 #1 Entry Bridle Roll 2 Drive Enable Safety Relay
        [0].30   // CHPLC:I.Data[1].6 x613CR710 #2 Entry Bridle Roll 3 Main Contactor Safety Relay
        [0].31   // CHPLC:I.Data[1].7 x613CR750 #2 Entry Bridle Roll 3 Drive Enable Safety Relay
        [1].0   // CHPLC:I.Data[2].0 x614CR040 #1 Exit Bridle Roll 6 Main Contactor Safety Relay
        [1].1   // CHPLC:I.Data[2].1 x614CR090 #1 Exit Bridle Roll 6 Drive Enable Safety Relay
        [1].2   // CHPLC:I.Data[2].2 x614CR130 #2 Exit Bridle Roll 7 Main Contactor Safety Relay
        [1].3   // CHPLC:I.Data[2].3 x614CR170 #2 Exit Bridle Roll 7 Drive Enable Safety Relay
        [1].4   // CHPLC:I.Data[2].4 x614CR210 Rewind Main Contactor Safety Relay
        [1].5   // CHPLC:I.Data[2].5 x614CR250 Rewind Drive Enable Safety Relay
        [1].6   // CHPLC:I.Data[2].6 CHPLC_S2_6 (SPARE)
        [1].7   // CHPLC:I.Data[2].7 CHPLC_S2_7 (SPARE)
        [1].8   // CHPLC:I.Data[3].0 CHPLC_S3_0 (SPARE)
        [1].9   // CHPLC:I.Data[3].1 CHPLC_S3_1 (SPARE)
        [1].10   // CHPLC:I.Data[3].2 CHPLC_S3_2 (SPARE)
        [1].11   // CHPLC:I.Data[3].3 CHPLC_S3_3 (SPARE)
        [1].12   // CHPLC:I.Data[3].4 CHPLC_S3_4 (SPARE)
        [1].13   // CHPLC:I.Data[3].5 CHPLC_S3_5 (SPARE)
        [1].14   // CHPLC:I.Data[3].6 CHPLC_S3_6 (SPARE)
        [1].15   // CHPLC:I.Data[3].7 CHPLC_S3_7 (SPARE)
        [1].16   // CHPLC:O.Data[4].0 y613CR460 Unwind Operator Side Main Contactor Safety Relay
        [1].17   // CHPLC:O.Data[4].1 y613CR510 Unwind Operator Side Drive Enable Safety Relay
        [1].18   // CHPLC:O.Data[4].2 y613CR550 Unwind Drive Side Main Contactor Safety Relay
        [1].19   // CHPLC:O.Data[4].3 y613CR590 Unwind Drive Side Drive Enable Safety Relay
        [1].20   // CHPLC:O.Data[4].4 y613CR630 #1 Entry Bridle Roll 2 Main Contactor Safety Relay
        [1].21   // CHPLC:O.Data[4].5 y613CR670 #1 Entry Bridle Roll 2 Drive Enable Safety Relay
        [1].22   // CHPLC:O.Data[4].6 y613CR710 #2 Entry Bridle Roll 3 Main Contactor Safety Relay
        [1].23   // CHPLC:O.Data[4].7 y613CR750 #2 Entry Bridle Roll 3 Drive Enable Safety Relay
        [1].24   // CHPLC:O.Data[5].0 y614CR040 #1 Exit Bridle Roll 6 Main Contactor Safety Relay
        [1].25   // CHPLC:O.Data[5].1 y614CR090 #1 Exit Bridle Roll 6 Drive Enable Safety Relay
        [1].26   // CHPLC:O.Data[5].2 y614CR130 #2 Exit Bridle Roll 7 Main Contactor Safety Relay
        [1].27   // CHPLC:O.Data[5].3 y614CR170 #2 Exit Bridle Roll 7 Drive Enable Safety Relay
        [1].28   // CHPLC:O.Data[5].4 y614CR210 Rewind Main Contactor Safety Relay
        [1].29   // CHPLC:O.Data[5].5 y614CR250 Rewind Drive Enable Safety Relay
        [1].30   // CHPLC:O.Data[5].6 CHPLC_S5_6 (SPARE)
        [1].31   // CHPLC:O.Data[5].7 CHPLC_S5_7 (SPARE)
        [2].0   // CHPLC:O.Data[6].0 CHPLC_S6_0 (SPARE)
        [2].1   // CHPLC:O.Data[6].1 CHPLC_S6_1 (SPARE)
        [2].2   // CHPLC:O.Data[6].2 CHPLC_S6_2 (SPARE)
        [2].3   // CHPLC:O.Data[6].3 CHPLC_S6_3 (SPARE)
        [2].4   // CHPLC:O.Data[6].4 CHPLC_S6_4 (SPARE)
        [2].5   // CHPLC:O.Data[6].5 CHPLC_S6_5 (SPARE)
        [2].6   // CHPLC:O.Data[6].6 CHPLC_S6_6 (SPARE)
        [2].7   // CHPLC:O.Data[6].7 CHPLC_S6_7 (SPARE)
        [2].8   // D1:O.Data[12].0 y451CR050 Soleniod Safe Off
        [2].9   // D1:O.Data[12].1 D1_S12_1 (SPARE)
        [2].10   // D1:O.Data[12].2 D1_S12_2 (SPARE)
        [2].11   // D1:O.Data[12].3 D1_S12_3 (SPARE)
        [2].12   // D1:O.Data[12].4 D1_S12_4 (SPARE)
        [2].13   // D1:O.Data[12].5 D1_S12_5 (SPARE)
        [2].14   // D1:O.Data[12].6 D1_S12_6 (SPARE)
        [2].15   // D1:O.Data[12].7 D1_S12_7 (SPARE)
        [2].16   // DPD:O.Data[14].0 y480CR050 Solenoid Safe Off
        [2].17   // DPD:O.Data[14].1 DPD_S14_1 (SPARE)
        [2].18   // DPD:O.Data[14].2 DPD_S14_2 (SPARE)
        [2].19   // DPD:O.Data[14].3 DPD_S14_3 (SPARE)
        [2].20   // DPD:O.Data[14].4 DPD_S14_4 (SPARE)
        [2].21   // DPD:O.Data[14].5 DPD_S14_5 (SPARE)
        [2].22   // DPD:O.Data[14].6 DPD_S14_6 (SPARE)
        [2].23   // DPD:O.Data[14].7 DPD_S14_7 (SPARE)
        [2].24   // DPD:I.Data[15].0 x480PB470a Emergency Stop Pushbutton
        [2].25   // DPD:I.Data[15].1 x480PB470b Emergency Stop Pushbutton
        [2].26   // DPD:I.Data[15].2 x480PB550a Emergency Stop Pushbutton (In Pit)
        [2].27   // DPD:I.Data[15].3 x480PB550b Emergency Stop Pushbutton (In Pit)
        [2].28   // DPD:I.Data[15].4 DPD_S15_4 (SPARE)
        [2].29   // DPD:I.Data[15].5 DPD_S15_5 (SPARE)
        [2].30   // DPD:I.Data[15].6 DPD_S15_6 (SPARE)
        [2].31   // DPD:I.Data[15].7 DPD_S15_7 (SPARE)
        [3].0   // E1:O.Data[10].0 y464CR050 Soleniod Safe Off
        [3].1   // E1:O.Data[10].1 E1_S10_1 (SPARE)
        [3].2   // E1:O.Data[10].2 E1_S10_2 (SPARE)
        [3].3   // E1:O.Data[10].3 E1_S10_3 (SPARE)
        [3].4   // E1:O.Data[10].4 E1_S10_4 (SPARE)
        [3].5   // E1:O.Data[10].5 E1_S10_5 (SPARE)
        [3].6   // E1:O.Data[10].6 E1_S10_6 (SPARE)
        [3].7   // E1:O.Data[10].7 E1_S10_7 (SPARE)
        [3].8   // F1:O.Data[19].0 y507CR050 Line Solenoid Safe Off
        [3].9   // F1:O.Data[19].1 y507CR090 Rewind Coil Car Solenoid Safe Off
        [3].10   // F1:O.Data[19].2 F1_S19_2 (SPARE)
        [3].11   // F1:O.Data[19].3 F1_S19_3 (SPARE)
        [3].12   // F1:O.Data[19].4 F1_S19_4 (SPARE)
        [3].13   // F1:O.Data[19].5 F1_S19_5 (SPARE)
        [3].14   // F1:O.Data[19].6 F1_S19_6 (SPARE)
        [3].15   // F1:O.Data[19].7 F1_S19_7 (SPARE)
        [3].16   // F1:I.Data[20].0 F1_S20_0 (SPARE)
        [3].17   // F1:I.Data[20].1 F1_S20_1 (SPARE)
        [3].18   // F1:I.Data[20].2 F1_S20_2 (SPARE)
        [3].19   // F1:I.Data[20].3 F1_S20_3 (SPARE)
        [3].20   // F1:I.Data[20].4 F1_S20_4 (SPARE)
        [3].21   // F1:I.Data[20].5 F1_S20_5 (SPARE)
        [3].22   // F1:I.Data[20].6 F1_S20_6 (SPARE)
        [3].23   // F1:I.Data[20].7 F1_S20_7 (SPARE)
        [3].24   // G1:O.Data[11].0 y519CR050 Line Solenoid Safe Off
        [3].25   // G1:O.Data[11].1 G1_S11_1 (SPARE)
        [3].26   // G1:O.Data[11].2 G1_S11_2 (SPARE)
        [3].27   // G1:O.Data[11].3 G1_S11_3 (SPARE)
        [3].28   // G1:O.Data[11].4 G1_S11_4 (SPARE)
        [3].29   // G1:O.Data[11].5 G1_S11_5 (SPARE)
        [3].30   // G1:O.Data[11].6 G1_S11_6 (SPARE)
        [3].31   // G1:O.Data[11].7 G1_S11_7 (SPARE)
        [4].0   // G1:I.Data[12].0 x519LS470 Tripwire Emergency Stop Limit Switch
        [4].1   // G1:I.Data[12].1 G1_S12_1 (SPARE)
        [4].2   // G1:I.Data[12].2 G1_S12_2 (SPARE)
        [4].3   // G1:I.Data[12].3 G1_S12_3 (SPARE)
        [4].4   // G1:I.Data[12].4 G1_S12_4 (SPARE)
        [4].5   // G1:I.Data[12].5 G1_S12_5 (SPARE)
        [4].6   // G1:I.Data[12].6 G1_S12_6 (SPARE)
        [4].7   // G1:I.Data[12].7 G1_S12_7 (SPARE)
        [4].8   // H1:O.Data[5].0 y533CR050 Line Solenoid Safe Off
        [4].9   // H1:O.Data[5].1 H1_S5_1 (SPARE)
        [4].10   // H1:O.Data[5].2 H1_S5_2 (SPARE)
        [4].11   // H1:O.Data[5].3 H1_S5_3 (SPARE)
        [4].12   // H1:O.Data[5].4 H1_S5_4 (SPARE)
        [4].13   // H1:O.Data[5].5 H1_S5_5 (SPARE)
        [4].14   // H1:O.Data[5].6 H1_S5_6 (SPARE)
        [4].15   // H1:O.Data[5].7 H1_S5_7 (SPARE)
        [4].16   // H1:I.Data[6].0 x533PB470a Sheeter Emergency Stop Pushbutton
        [4].17   // H1:I.Data[6].1 x533PB470b Sheeter Emergency Stop Pushbutton
        [4].18   // H1:I.Data[6].2 H1_S6_2 (SPARE)
        [4].19   // H1:I.Data[6].3 H1_S6_3 (SPARE)
        [4].20   // H1:I.Data[6].4 H1_S6_4 (SPARE)
        [4].21   // H1:I.Data[6].5 H1_S6_5 (SPARE)
        [4].22   // H1:I.Data[6].6 H1_S6_6 (SPARE)
        [4].23   // H1:I.Data[6].7 H1_S6_7 (SPARE)
        [4].24   // MCC1:I.Data[1].0 x702MTR191FF Rewind Pinch Roll Fwd Fdbk
        [4].25   // MCC1:I.Data[1].1 x702MTR191RF Rewind Pinch Roll Rev Fdbk
        [4].26   // MCC1:I.Data[1].2 MCC1_S1_2 (SPARE)
        [4].27   // MCC1:I.Data[1].3 MCC1_S1_3 (SPARE)
        [4].28   // MCC1:I.Data[1].4 x708MTR080FF Flattener Drive Motor Fwd Fdbk
        [4].29   // MCC1:I.Data[1].5 x708MTR080RF Flattener Drive Motor Rev Fdbk
        [4].30   // MCC1:I.Data[1].6 x708MTR250FF Unwind Holddown Roll Drive Motor Fwd Fdbk
        [4].31   // MCC1:I.Data[1].7 x708MTR250RF Unwind Holddown Roll Drive Motor Rev Fdbk
        [5].0   // MCC1:O.Data[6].0 y702MTR191FC Rewind Pinch Roll Fwd Cmd
        [5].1   // MCC1:O.Data[6].1 y702MTR191RC Rewind Pinch Roll Rev Cmd
        [5].2   // MCC1:O.Data[6].2 MCC1_S6_2 (SPARE)
        [5].3   // MCC1:O.Data[6].3 MCC1_S6_3 (SPARE)
        [5].4   // MCC1:O.Data[6].4 y708MTR080FC Flattener Drive Motor Fwd Cmd
        [5].5   // MCC1:O.Data[6].5 y708MTR080RC Flattener Drive Motor Rev Cmd
        [5].6   // MCC1:O.Data[6].6 y708MTR250FC Unwind Holddown Roll Drive Motor Fwd Cmd
        [5].7   // MCC1:O.Data[6].7 y708MTR250RC Unwind Holddown Roll Drive Motor Rev Cmd
        [5].8   // MCC2:O.Data[1].0 y725MTR080SP Unwind Pinch Roll Safety Power
        [5].9   // MCC2:O.Data[1].1 y725MTR080SE Unwind Pinch Roll Safety Enable
        [5].10   // MCC2:O.Data[1].2 y729MTR080SP Washtank Pinch Roll 4 Safety Power
        [5].11   // MCC2:O.Data[1].3 y729MTR080SE Washtank Pinch Roll 4 Safety Enable
        [5].12   // MCC2:O.Data[1].4 y727MTR080SP Paper Winder Safety Power
        [5].13   // MCC2:O.Data[1].5 y727MTR080SE Paper Winder Safety Enable
        [5].14   // MCC2:O.Data[1].6 y731MTR080SP Washtank Pinch Roll 1 Safety Power
        [5].15   // MCC2:O.Data[1].7 y731MTR080SE Washtank Pinch Roll 1 Safety Enable
        [5].16   // MCC2:O.Data[2].0 y733MTR080SP Washtank Pinch Roll 2 Safety Power
        [5].17   // MCC2:O.Data[2].1 y733MTR080SE Washtank Pinch Roll 2 Safety Enable
        [5].18   // MCC2:O.Data[2].2 y735MTR080SP Washtank Pinch Roll 3 Safety Power
        [5].19   // MCC2:O.Data[2].3 y735MTR080SE Washtank Pinch Roll 3 Safety Enable
        [5].20   // MCC2:O.Data[2].4 MCC2_S2_4 (SPARE)
        [5].21   // MCC2:O.Data[2].5 MCC2_S2_5 (SPARE)
        [5].22   // MCC2:O.Data[2].6 MCC2_S2_6 (SPARE)
        [5].23   // MCC2:O.Data[2].7 MCC2_S2_7 (SPARE)
        [5].24   // MCC3:I.Data[1].0 x753MTR190FF Trimmer Pinch Roll Fwd Fdbk
        [5].25   // MCC3:I.Data[1].1 x753MTR190RF Trimmer Pinch Roll Rev Fdbk
        [5].26   // MCC3:I.Data[1].2 x761MTR081RF Trimmer Scrap Conveyor RunFdbk
        [5].27   // MCC3:I.Data[1].3 MCC3_S1_3 (SPARE)
        [5].28   // MCC3:I.Data[1].4 MCC3_S1_4 (SPARE)
        [5].29   // MCC3:I.Data[1].5 MCC3_S1_5 (SPARE)
        [5].30   // MCC3:I.Data[1].6 MCC3_S1_6 (SPARE)
        [5].31   // MCC3:I.Data[1].7 MCC3_S1_7 (SPARE)
        [6].0   // MCC3:O.Data[3].0 y753MTR190FC Trimmer Pinch Roll Fwd Cmd
        [6].1   // MCC3:O.Data[3].1 y753MTR190RC Trimmer Pinch Roll Rev Cmd
        [6].2   // MCC3:O.Data[3].2 y761MTR081RC Trimmer Scrap Conveyor RunCmd
        [6].3   // MCC3:O.Data[3].3 y751MTR080SP Trimmer Knives Safety Power
        [6].4   // MCC3:O.Data[3].4 y751MTR080SE Trimmer Knives Safety Enable
        [6].5   // MCC3:O.Data[3].5 y754MTR080SP Side Guide Width Adjust Safety Power
        [6].6   // MCC3:O.Data[3].6 y754MTR080SE Side Guide Width Adjust Safety Enable
        [6].7   // MCC3:O.Data[3].7 y755MTR080SP Trimmer Knives Width Adjust Safety Power
        [6].8   // MCC3:O.Data[4].0 y755MTR080SE Trimmer Knives Width Adjust Safety Enable
        [6].9   // MCC3:O.Data[4].1 x759MTR080SP Scrap Choppers Width Adjust Safety Power
        [6].10   // MCC3:O.Data[4].2 x759MTR080SE Scrap Choppers Width Adjust Safety Enable
        [6].11   // MCC3:O.Data[4].3 y762MTR080SP Scrap Choppers Safety Power
        [6].12   // MCC3:O.Data[4].4 y762MTR080SE Scrap Choppers Safety Enable
        [6].13   // MCC3:O.Data[4].5 MCC3_S4_5 (SPARE)
        [6].14   // MCC3:O.Data[4].6 MCC3_S4_6 (SPARE)
        [6].15   // MCC3:O.Data[4].7 MCC3_S4_7 (SPARE)
        [6].16   // MCC4:I.Data[1].0 x778MTR080RF Shear Crank Motor Run Fdbk
        [6].17   // MCC4:I.Data[1].1 MCC4_S1_1 (SPARE)
        [6].18   // MCC4:I.Data[1].2 MCC4_S1_2 (SPARE)
        [6].19   // MCC4:I.Data[1].3 MCC4_S1_3 (SPARE)
        [6].20   // MCC4:I.Data[1].4 MCC4_S1_4 (SPARE)
        [6].21   // MCC4:I.Data[1].5 MCC4_S1_5 (SPARE)
        [6].22   // MCC4:I.Data[1].6 MCC4_S1_6 (SPARE)
        [6].23   // MCC4:I.Data[1].7 MCC4_S1_7 (SPARE)
        [6].24   // MCC4:O.Data[3].0 y779MTR080SP Shear Pinch Roll Safety Power
        [6].25   // MCC4:O.Data[3].1 y779MTR080SE Shear Pinch Roll Safety Enable
        [6].26   // MCC4:O.Data[3].2 y782MTR080SP Sheeter Pinch Roll Safety Power
        [6].27   // MCC4:O.Data[3].3 y782MTR080SE Sheeter Pinch Roll Safety Enable
        [6].28   // MCC4:O.Data[3].4 y785MTR080SP Stacker Blower Safety Power
        [6].29   // MCC4:O.Data[3].5 y785MTR080SE Stacker Blower Safety Enable
        [6].30   // MCC4:O.Data[3].6 y776MTR080SP Shear Metering Backup Roll Safety Power
        [6].31   // MCC4:O.Data[3].7 y776MTR080SE Shear Metering Backup Roll Safety Enable
        [7].0   // MCC4:O.Data[4].0 y778MTR080RC Shear Die Crank Run Cmd
        [7].1   // MCC4:O.Data[4].1 MCC4_S4_1 (SPARE)
        [7].2   // MCC4:O.Data[4].2 MCC4_S4_2 (SPARE)
        [7].3   // MCC4:O.Data[4].3 MCC4_S4_3 (SPARE)
        [7].4   // MCC4:O.Data[4].4 MCC4_S4_4 (SPARE)
        [7].5   // MCC4:O.Data[4].5 MCC4_S4_5 (SPARE)
        [7].6   // MCC4:O.Data[4].6 MCC4_S4_6 (SPARE)
        [7].7   // MCC4:O.Data[4].7 MCC4_S4_7 (SPARE)
        [7].8   // MCC5:I.Data[1].0 x802MTR080FF Stacker Side Guide Lift Fwd Fdbk/Up
        [7].9   // MCC5:I.Data[1].1 x802MTR080RF Stacker Side Guide Lift Rev Fdbk/Down
        [7].10   // MCC5:I.Data[1].2 x802MTR230FF Scrap Horizontal Conveyor Run Fwd Fdbk
        [7].11   // MCC5:I.Data[1].3 x802MTR230RF Scrap Horizontal Conveyor Run Rev Fdbk
        [7].12   // MCC5:I.Data[1].4 x802MTR231FF Stacker Chain Fwd Fdbk
        [7].13   // MCC5:I.Data[1].5 x802MTR231RF Stacker Chain Rev Fdbk
        [7].14   // MCC5:I.Data[1].6 MCC5_S1_6 (SPARE)
        [7].15   // MCC5:I.Data[1].7 MCC5_S1_7 (SPARE)
        [7].16   // MCC5:O.Data[3].0 y800MTR080SP Scrap Incline Conveyor Safety Power
        [7].17   // MCC5:O.Data[3].1 y800MTR080SE Scrap Incline Conveyor Safety Enable
        [7].18   // MCC5:O.Data[3].2 y804MTR080SP Stacker Back Stop Safety Power
        [7].19   // MCC5:O.Data[3].3 y804MTR080SE Stacker Back Stop Safety Enable
        [7].20   // MCC5:O.Data[3].4 y806MTR080SP Product Conveyor 3 Safety Power
        [7].21   // MCC5:O.Data[3].5 y806MTR080SE Product Conveyor 3 Safety Enable
        [7].22   // MCC5:O.Data[3].6 y808MTR080SP Product Conveyor 1 Safety Power
        [7].23   // MCC5:O.Data[3].7 y808MTR080SE Product Conveyor 1 Safety Enable
        [7].24   // MCC5:O.Data[4].0 y810MTR080SP Product Conveyor 2 Safety Power
        [7].25   // MCC5:O.Data[4].1 y810MTR080SE Product Conveyor 2 Safety Enable
        [7].26   // MCC5:O.Data[4].2 y812MTR080SP Shear Conveyor Safety Power
        [7].27   // MCC5:O.Data[4].3 y812MTR080SE Shear Conveyor Safety Enable
        [7].28   // MCC5:O.Data[4].4 y802MTR080FC Stacker Side Guide Lift Fwd Cmd/Up
        [7].29   // MCC5:O.Data[4].5 y802MTR080RC Stacker Side Guide Lift Rev Cmd/Down
        [7].30   // MCC5:O.Data[4].6 y802MTR230FC Scrap Horizontal Conveyor Fwd Cmd
        [7].31   // MCC5:O.Data[4].7 y802MTR230RC Scrap Horizontal Conveyor Rev Cmd
        [8].0   // MCC5:O.Data[5].0 y802MTR231FC Stacker Chain Fwd Cmd
        [8].1   // MCC5:O.Data[5].1 y802MTR231RC Stacker Chain Rev Cmd
        [8].2   // MCC5:O.Data[5].2 MCC5_S5_2 (SPARE)
        [8].3   // MCC5:O.Data[5].3 MCC5_S5_3 (SPARE)
        [8].4   // MCC5:O.Data[5].4 MCC5_S5_4 (SPARE)
        [8].5   // MCC5:O.Data[5].5 MCC5_S5_5 (SPARE)
        [8].6   // MCC5:O.Data[5].6 MCC5_S5_6 (SPARE)
        [8].7   // MCC5:O.Data[5].7 MCC5_S5_7 (SPARE)
        [8].8   // SDPLC:I.Data[1].0 x172CR460 Shear Die Drive Main Contactor Safety Relay Input
        [8].9   // SDPLC:I.Data[1].1 x172CR510 Shear Die Drive Enable Safety Relay Input
        [8].10   // SDPLC:I.Data[1].2 SDPLC_S1_2 (SPARE)
        [8].11   // SDPLC:I.Data[1].3 SDPLC_S1_3 (SPARE)
        [8].12   // SDPLC:I.Data[1].4 SDPLC_S1_4 (SPARE)
        [8].13   // SDPLC:I.Data[1].5 SDPLC_S1_5 (SPARE)
        [8].14   // SDPLC:I.Data[1].6 SDPLC_S1_6 (SPARE)
        [8].15   // SDPLC:I.Data[1].7 SDPLC_S1_7 (SPARE)
        [8].16   // SDPLC:O.Data[2].0 y172CR460 Shear Die Drive Main Contactor Safety Relay Output
        [8].17   // SDPLC:O.Data[2].1 y172CR510 Shear Die Drive Enable Safety Relay Output
        [8].18   // SDPLC:O.Data[2].2 y172CR550 Line Soleniod Safe-Off
        [8].19   // SDPLC:O.Data[2].3 SDPLC_S2_2 (SPARE)
        [8].20   // SDPLC:O.Data[2].4 SDPLC_S2_3 (SPARE)
        [8].21   // SDPLC:O.Data[2].5 SDPLC_S2_4 (SPARE)
        [8].22   // SDPLC:O.Data[2].6 SDPLC_S2_5 (SPARE)
        [8].23   // SDPLC:O.Data[2].7 SDPLC_S2_6 (SPARE)
   TrimPR_FVR_En : BOOL := 1;   // Trimmer Pinch Roll FVR Enable ( 1= Enable )
   TrimPR_FVR_FltRst : BOOL;   // Trimmer Pinch Roll Fault Reset ( 1= Reset Cmd )
   TrimPR_FVR_FwdCmd : BOOL;   // Trimmer Pinch Roll Forward Command ( 1= Run Fwd )
   TrimPR_FVR_RevCmd : BOOL;   // Trimmer Pinch Roll Reverse Command ( 1= Run Rev)
   TrimScCon_FVNR_En : BOOL := 1;   // Trimmer Scrap Conveyor FVNR Enable ( 1= Enable )
   TrimScCon_FVNR_FltRst : BOOL;   // Trimmer Scrap Conveyor Fault Reset ( 1= Reset Cmd )
   TrimScCon_FVNR_RunCmd : BOOL := 1;   // Trimmer Scrap Conveyor Run Command ( 1= Run )
   UnPR_DrvsOff : BOOL;   // Unwind Pinch Roll Drives OFF ( 1= OFF)
   UnPR_SafeTrqEn : BOOL := 1;   // Unwind Pinch Roll Safe-Trq Off Enable ( 1= Enable )
   UNW_DrvsOff : BOOL;   // Unwind Drives OFF ( 1= OFF)
   UNW_SafeOffEn : BOOL := 1;   // Unwind Safe-Off Enable ( 1= Enable )
